Omron CX-Programmer project 新規ﾌﾟﾛｼﾞｪｸﾄ (CX-Programmer 9.34)

# PLC DCS_PLC: CJ2M CPU13
I/O table (CPU CJ2M-CPU13): rack 0 slot 0 CJ1W-CLK23; rack 0 slot 1 CJ1W-SCU21-V1; rack 0 slot 2 CJ1W-OD211

## Global symbols (name address type ; comment)
0.05 BOOL  ; error_clear_sw
12 CHANNEL  ; CH1PV１次1,2桁目
1534.06 BOOL  ; P1受信完了ﾌﾗｸﾞ
1544.06 BOOL  ; P2受信完了ﾌﾗｸﾞ
1559.05 BOOL  ; TXDU命令実行中ﾌﾗｸﾞ
1634.06 BOOL  ; -
2.10 BOOL  ; lot_trace_camera_out1
2.11 BOOL  ; lot_trace_camera_out2
2.12 BOOL  ; lot_trace_camera_out3
2.13 BOOL  ; lot_trace_camera_out4
3000.01 BOOL  ; 送り
3000.02 BOOL  ; 全検査完了
3000.03 BOOL  ; 装置再投入フラグ
3010.01 BOOL  ; ﾗﾝﾆﾝｸﾞ_disable
3010.02 BOOL  ; 耐圧CC_disable
3010.03 BOOL  ; 耐圧CF_disable
3010.04 BOOL  ; 有負荷disable
3010.05 BOOL  ; ｲﾝﾊﾟﾙｽ_disable
3010.06 BOOL  ; ｵﾌﾊﾞｳﾝｽ_disable
3010.07 BOOL  ; RT_disable
3010.08 BOOL  ; MVD_disable
3020.06 BOOL  ; R1_OK
3020.07 BOOL  ; R2_OK
3020.08 BOOL  ; R3_OK
3020.09 BOOL  ; R4_OK
3020.10 BOOL  ; R5_OK
3020.11 BOOL  ; R6_OK
3020.12 BOOL  ; R7_OK
3020.13 BOOL  ; R8_OK
3020.14 BOOL  ; R9_OK
3020.15 BOOL  ; R10_OK
3021.00 BOOL  ; 耐圧CC_OK
3021.01 BOOL  ; 耐圧CF_OK
3021.02 BOOL  ; ｲﾝﾊﾟﾙｽ_OK
3021.03 BOOL  ; 有負荷_OK
3021.04 BOOL  ; ｵﾌﾊﾞｳﾝｽ_OK
3021.05 BOOL  ; RT_OK
3021.06 BOOL  ; MVD_OK
3022.06 BOOL  ; R1_NG
3022.07 BOOL  ; R2_NG
3022.08 BOOL  ; R3_NG
3022.09 BOOL  ; R4_NG
3022.10 BOOL  ; R5_NG
3022.11 BOOL  ; R6_NG
3022.12 BOOL  ; R7_NG
3022.13 BOOL  ; R8_OK
3022.14 BOOL  ; R9_OK
3022.15 BOOL  ; R10_OK
3023.00 BOOL  ; 耐圧CC_OK
3023.01 BOOL  ; 耐圧CF_OK
3023.02 BOOL  ; ｲﾝﾊﾟﾙｽ_OK
3023.03 BOOL  ; 有負荷_OK
3023.04 BOOL  ; ｵﾌﾊﾞｳﾝｽ_OK
3023.05 BOOL  ; RT_OK
3023.06 BOOL  ; MVD_OK
3024.00 BOOL  ; R1
3024.01 BOOL  ; R2
3024.02 BOOL  ; R3
3024.03 BOOL  ; R4
3024.04 BOOL  ; R5
3024.05 BOOL  ; R6
3024.06 BOOL  ; R7
3024.07 BOOL  ; R8
3024.08 BOOL  ; R9
3024.09 BOOL  ; ﾗﾝﾆﾝｸﾞ
3024.10 BOOL  ; 耐圧C-F
3024.11 BOOL  ; 耐圧C-C
3024.12 BOOL  ; ｺｲﾙｲﾝﾊﾟﾙｽ
3024.13 BOOL  ; 有負荷ﾗﾝﾆﾝｸﾞ
3024.14 BOOL  ; ｵﾌﾊﾞｳﾝｽ
3024.15 BOOL  ; CIR
3025.00 BOOL  ; PV-H
3025.01 BOOL  ; PV-L
3025.02 BOOL  ; DV-H
3025.03 BOOL  ; DV-L
3025.04 BOOL  ; TSO
3025.05 BOOL  ; MVD
3050.00 BOOL  ; Ready_RT
3050.01 BOOL  ; Ready_CP
3100.00 BOOL  ; ﾃﾞｰﾀ収集Home
3100.01 BOOL  ; ﾃﾞｰﾀ収集FULL
3100.02 BOOL  ; ﾃﾞｰﾀ収集Ready
3100.03 BOOL  ; CP繰返測定モード
3228 CHANNEL  ; Z2_Target_position
3328 CHANNEL  ; Z2_Now_position
4.14 BOOL  ; lot_trace_camera_out
5000.00 BOOL  ; ﾃﾞｰﾀ収集PLC原点OK
5000.01 BOOL  ; ﾃﾞｰﾀﾊﾞｯﾌｧｰFull
5000.02 BOOL  ; ﾃﾞｰﾀ収集Ready
500.01 BOOL  ; 取出
902.11 BOOL  ; tp_delate_sw
902.12 BOOL  ; tp_all_delete_yes_sw
A202.00 BOOL  ; ﾈｯﾄﾜｰｸ通信命令実行可ﾌﾗｸﾞ
A351 CHANNEL  ; 分秒
A352 CHANNEL  ; 日時
A353 CHANNEL  ; 年月
A356.05 BOOL  ; PORT1送信ﾚﾃﾞｲﾌﾗｸﾞ
A392.05 BOOL  ; RS232Cﾎﾟｰﾄ送信ﾚﾃﾞｲﾌﾗｸﾞ
D0 CHANNEL  ; PC心拍数
D1 CHANNEL  ; PC心拍ﾃﾞｸﾘﾒﾝﾄ用ﾌﾟﾘｽｹｰﾗ
D10 CHANNEL  ; 結果ﾃﾞｰﾀ
D100 CHANNEL  ; 受信CH1PV1,2桁
D1000 CHANNEL  ; １ﾊﾞｲﾄ目
D10000 CHANNEL  ; 1ST
D10000.00 BOOL  ; 搬送送りﾄﾘｶﾞ
D10001.00 BOOL  ; 搬送RT1検査実施
D10001.01 BOOL  ; 搬送RT2検査実施
D10001.02 BOOL  ; 搬送RT3検査実施
D10001.03 BOOL  ; 搬送CP1検査実施
D10001.04 BOOL  ; 搬送CP2検査実施
D10001.05 BOOL  ; 搬送CP3検査実施
D10002.00 BOOL  ; 搬送検査ﾄﾘｶﾞ
D1000.00 BOOL  ; 搬送PLCﾃﾞｰﾀ出力ﾄﾘｶﾞ
D10010 CHANNEL  ; PF_Ch1OVL
D10011 CHANNEL  ; PF_Ch1OVR
D10012 CHANNEL  ; PV_IN
D10014 CHANNEL  ; DV_IN
D10016 CHANNEL  ; CIR_IN
D10018 CHANNEL  ; TSO_IN
D10028 CHANNEL  ; NC_IN
D10030 CHANNEL  ; NO_IN
D10032 CHANNEL  ; CG_IN
D10040 CHANNEL  ; PF_Ch3TOL
D10041 CHANNEL  ; PF_Ch3TOR
D101 CHANNEL  ; 受信CH1PV3,4桁
D10128 CHANNEL  ; NC_IN
D10130 CHANNEL  ; NO_IN
D10132 CHANNEL  ; CG_IN
D102 CHANNEL  ; 受信CH1PV5桁目と小数点
D10200 CHANNEL  ; 3ST
D10202 CHANNEL  ; R2_IN
D10212 CHANNEL  ; PV_OUT
D10214 CHANNEL  ; DV_OUT
D10216 CHANNEL  ; CIR_OUT
D10218 CHANNEL  ; TSO_OUT
D10228 CHANNEL  ; NC_IN
D10230 CHANNEL  ; NO_IN
D10232 CHANNEL  ; CG_OUT
D103 CHANNEL  ; 受信CH1PV6,7桁目
D10300 CHANNEL  ; 4ST
D10303 CHANNEL  ; R3_IN
D10312 CHANNEL  ; PV_OUT
D10314 CHANNEL  ; DV_OUT
D10316 CHANNEL  ; CIR_OUT
D10318 CHANNEL  ; TSO_OUT
D10328 CHANNEL  ; NC_OUT
D10330 CHANNEL  ; NO_OUT
D10332 CHANNEL  ; CG_OUT
D104 CHANNEL  ; 受信CH1DVt,1桁目
D10400 CHANNEL  ; 5ST
D10404 CHANNEL  ; R4_IN
D10412 CHANNEL  ; PV_OUT
D10414 CHANNEL  ; DV_OUT
D10416 CHANNEL  ; CIR_OUT
D10418 CHANNEL  ; TSO_OUT
D10428 CHANNEL  ; NC_OUT
D10430 CHANNEL  ; NO_OUT
D10432 CHANNEL  ; CG_OUT
D105 CHANNEL  ; 受信CH1DV2,3桁目
D10500 CHANNEL  ; 6ST
D10505 CHANNEL  ; R5_IN
D106 CHANNEL  ; 受信CH1DV4,5桁目
D10600 CHANNEL  ; 7ST
D107 CHANNEL  ; 受信CH1DV小数点と6桁目
D10700 CHANNEL  ; 8ST
D10707 CHANNEL  ; 耐圧CC_IN
D108 CHANNEL  ; 受信CH1DV7桁目とt
D10800 CHANNEL  ; 9ST
D10808 CHANNEL  ; 耐圧CF_IN
D109 CHANNEL  ; 受信CH1ｺｲﾙR1,2桁目
D10900 CHANNEL  ; 10ST
D10909 CHANNEL  ; ｲﾝﾊﾟﾙｽIN
D110 CHANNEL  ; 受信CH1ｺｲﾙR3,4桁目
D1100 CHANNEL  ; 結果
D11000 CHANNEL  ; 送信ｴﾘｱ収集PLC
D11010 CHANNEL  ; 有負荷IN
D111 CHANNEL  ; 受信CH1ｺｲﾙR5,6桁目
D11100 CHANNEL  ; 12ST
D11111 CHANNEL  ; ｵﾌﾊﾞｳﾝｽ_IN
D112 CHANNEL  ; 受信CH1ｺｲﾙR小数点,7桁目
D11200 CHANNEL  ; 13ST
D11212 CHANNEL  ; PV_IN
D11214 CHANNEL  ; DV_IN
D11216 CHANNEL  ; CIR_IN
D11218 CHANNEL  ; TSO_IN
D11228 CHANNEL  ; MVD_IN
D11300 CHANNEL  ; 14ST
D11328 CHANNEL  ; MVD_IN
D114 CHANNEL  ; 受信CH1TSO2,3桁目
D11400 CHANNEL  ; 15ST
D115 CHANNEL  ; 受信CH1TSO4,5桁目
D11500 CHANNEL  ; 16ST
D11531 CHANNEL  ; R6_IN
D116 CHANNEL  ; 受信CH1TSO小数点6桁目
D11600 CHANNEL  ; 17ST
D11632 CHANNEL  ; R7_IN
D117 CHANNEL  ; 受信CH1TSO7桁目,t
D11700 CHANNEL  ; 18ST
D11733 CHANNEL  ; R8_IN
D11800 CHANNEL  ; 19ST
D11834 CHANNEL  ; R9_IN
D11900 CHANNEL  ; 20ST
D11935 CHANNEL  ; R10_IN
D11996.00 BOOL  ; 収集PLCﾃﾞｰﾀ満杯
D11997.00 BOOL  ; PC起動OKﾌﾗｸﾞ
D11998 CHANNEL  ; PC読込許可ﾌﾗｸﾞ
D11999 CHANNEL  ; PC読込完了ﾌﾗｸﾞｸﾘｱ依頼
D12000 CHANNEL  ; PC読込完了ﾌﾗｸﾞ
D12001.00 BOOL  ; PC起動中Pulse
D12100 CHANNEL  ; 22ST
D12200 CHANNEL  ; 23ST
D12212 CHANNEL  ; PV_OUT
D12300 CHANNEL  ; 24ST
D12400 CHANNEL  ; 25ST
D12401 CHANNEL  ; R1_OUT
D12402 CHANNEL  ; R2_OUT
D12403 CHANNEL  ; R3_OUT
D12404 CHANNEL  ; R4_OUT
D12405 CHANNEL  ; R5_OUT
D12407 CHANNEL  ; 耐圧CC_OUT
D12408 CHANNEL  ; 耐圧CF_OUT
D12409 CHANNEL  ; ｲﾝﾊﾟﾙｽOUT
D12410 CHANNEL  ; 有負荷OUT
D12411 CHANNEL  ; ｵﾌﾊﾞｳﾝｽ_OUT
D12412 CHANNEL  ; PV_OUT
D12414 CHANNEL  ; DV_OUT
D12416 CHANNEL  ; CIR_OUT
D12418 CHANNEL  ; TSO_OUT
D12428 CHANNEL  ; MVD_OUT
D12431 CHANNEL  ; R6_OUT
D12432 CHANNEL  ; R7_OUT
D12433 CHANNEL  ; R8_OUT
D12434 CHANNEL  ; R9_OUT
D12435 CHANNEL  ; R10_OUT
D12500 CHANNEL  ; 26ST
D12600 CHANNEL  ; 27ST
D12700 CHANNEL  ; 28ST
D12701 CHANNEL  ; R1_OUT
D12702 CHANNEL  ; R2_OUT
D12703 CHANNEL  ; R3_OUT
D12704 CHANNEL  ; R4_OUT
D12705 CHANNEL  ; R5_OUT
D12707 CHANNEL  ; 耐圧CC_OUT
D12708 CHANNEL  ; 耐圧CF_OUT
D12709 CHANNEL  ; ｲﾝﾊﾟﾙｽOUT
D12710 CHANNEL  ; 有負荷OUT
D12711 CHANNEL  ; ｵﾌﾊﾞｳﾝｽOUT
D12712 CHANNEL  ; PV_OUT
D12714 CHANNEL  ; DV_OUT
D12716 CHANNEL  ; CIR_OUT
D12718 CHANNEL  ; TSO_OUT
D12728 CHANNEL  ; MVD_OUT
D12730 CHANNEL  ; NO_OUT
D12731 CHANNEL  ; R6_OUT
D12732 CHANNEL  ; R7_OUT
D12733 CHANNEL  ; R8_OUT
D12734 CHANNEL  ; R9_OUT
D12735 CHANNEL  ; R10_OUT
D13000 CHANNEL  ; TMP有無
D13001 CHANNEL  ; TMP分秒
D13002 CHANNEL  ; TMP日時
D13003 CHANNEL  ; TMP年月
D13004 CHANNEL  ; TMP順番
D13005 CHANNEL  ; TMPﾁｬﾝﾈﾙ
D13006 CHANNEL  ; TMPﾁｬﾝﾈﾙ
D13007 CHANNEL  ; TMP機種コード
D13008 CHANNEL  ; TMP機種名
D13018 CHANNEL  ; TMP再投入
D13019 CHANNEL  ; PV_TMP
D13021 CHANNEL  ; DV_TMP
D13023 CHANNEL  ; TSO_TMP
D13025 CHANNEL  ; NC_TMP
D13027 CHANNEL  ; NO_TMP
D13029 CHANNEL  ; CG_TMP
D13031 CHANNEL  ; PV_TMP
D13033 CHANNEL  ; DV_TMP
D13035 CHANNEL  ; TSO_TMP
D13037 CHANNEL  ; CIR_TMP
D13039 CHANNEL  ; MVD_TMP
D13041 CHANNEL  ; 有負荷R_TMP
D13042 CHANNEL  ; 耐圧C-F_TMP
D13043 CHANNEL  ; 耐圧C-C_TMP
D13044 CHANNEL  ; ｵﾌﾊﾞｳﾝｽ_TMP
D13045 CHANNEL  ; ｲﾝﾊﾟﾙｽ_TMP
D13046 CHANNEL  ; ﾗﾝﾆﾝｸﾞ_TMP
D13047 CHANNEL  ; TMP判定
D13050 CHANNEL  ; PV_TMP
D13052 CHANNEL  ; DV_TMP
D13054 CHANNEL  ; TSO_TMP
D13056 CHANNEL  ; CIR_TMP
D13058 CHANNEL  ; NC_MVD_TMP
D13060 CHANNEL  ; NO_TMP
D13062 CHANNEL  ; CG_IN
D13063 CHANNEL  ; 有負荷_TMP
D13064 CHANNEL  ; 耐圧CC_TMP
D13065 CHANNEL  ; 耐圧CF_TMP
D13066 CHANNEL  ; ｵﾌﾊﾞｳﾝｽ_TMP
D13067 CHANNEL  ; ｲﾝﾊﾟﾙｽ_TMP
D13068 CHANNEL  ; R1TMP
D13069 CHANNEL  ; R2_TMP
D13070 CHANNEL  ; R3_TMP
D13071 CHANNEL  ; R4_TMP
D13072 CHANNEL  ; R5_TMP
D13073 CHANNEL  ; R6_TMP
D13074 CHANNEL  ; R7_TMP
D13075 CHANNEL  ; R8_TMP
D13076 CHANNEL  ; R9_TMP
D13077 CHANNEL  ; R10_TMP
D13078 CHANNEL  ; RT_TMP
D13079 CHANNEL  ; MVD_TMP
D13100 CHANNEL  ; PC書込中フラグ
D13102 CHANNEL  ; ﾃﾞﾊﾞｯｸﾞ用カウンタ
D13200 CHANNEL  ; Dｴﾘｱｸﾘｱﾎﾟｲﾝﾀ
D13300 CHANNEL  ; ｺﾝﾄﾛｰﾙﾃﾞｰﾀ1-1
D13301 CHANNEL  ; ｺﾝﾄﾛｰﾙﾃﾞｰﾀ1-2
D13302 CHANNEL  ; ｺﾝﾄﾛｰﾙﾃﾞｰﾀ2-1
D13303 CHANNEL  ; ｺﾝﾄﾛｰﾙﾃﾞｰﾀ2-2
D13400 CHANNEL  ; RT受信ﾃﾞｰﾀ1
D13402 CHANNEL  ; RT受信ﾃﾞｰﾀPV3
D13403 CHANNEL  ; RT受信ﾃﾞｰﾀ2
D13404 CHANNEL  ; RT受信ﾃﾞｰﾀDV4
D13405 CHANNEL  ; RT受信ﾃﾞｰﾀDV1
D13406 CHANNEL  ; RT受信ﾃﾞｰﾀ3
D13407 CHANNEL  ; RT受信ﾃﾞｰﾀDV3
D13408 CHANNEL  ; RT受信ﾃﾞｰﾀDV3
D13409 CHANNEL  ; RT受信ﾃﾞｰﾀ4
D13410 CHANNEL  ; RT受信ﾃﾞｰﾀCI2
D13411 CHANNEL  ; RT受信ﾃﾞｰﾀCI3
D13412 CHANNEL  ; RT受信ﾃﾞｰﾀ5
D13414 CHANNEL  ; RT受信ﾃﾞｰﾀTSO1
D13415 CHANNEL  ; RT受信ﾃﾞｰﾀ6
D13416 CHANNEL  ; RT受信ﾃﾞｰﾀTSO3
D13417 CHANNEL  ; RT受信ﾃﾞｰﾀTSO4
D13450 CHANNEL  ; RT_OVL
D13452 CHANNEL  ; RT_OVR
D13453 CHANNEL  ; PV1次4
D13454 CHANNEL  ; RT_RVL
D13455 CHANNEL  ; DV1次1
D13456 CHANNEL  ; RT_RVR
D13457 CHANNEL  ; DV1次3
D13458 CHANNEL  ; DV1次4
D13460 CHANNEL  ; CP_Ch1NCL
D13461 CHANNEL  ; CI1次2
D13462 CHANNEL  ; CP_Ch1NCR
D13463 CHANNEL  ; CI1次4
D13464 CHANNEL  ; CP_Ch1NOL
D13465 CHANNEL  ; TSO1次1
D13466 CHANNEL  ; CP_Ch1NOR
D13467 CHANNEL  ; TSO1次3
D13468 CHANNEL  ; CP_Ch1CGL
D13469 CHANNEL  ; CI1次5
D13470 CHANNEL  ; CP_Ch1CGR
D13472 CHANNEL  ; CP_Ch2NCL
D13474 CHANNEL  ; CP_Ch2NCR
D13476 CHANNEL  ; CP_Ch2NOL
D13478 CHANNEL  ; CP_Ch2NOR
D13480 CHANNEL  ; CP_Ch2CGL
D13482 CHANNEL  ; CP_Ch2CGR
D13484 CHANNEL  ; CP_Ch3NCL
D13486 CHANNEL  ; CP_Ch3NCR
D13488 CHANNEL  ; CP_Ch3NOL
D13490 CHANNEL  ; CP_Ch3NOR
D13492 CHANNEL  ; CP_Ch3CGL
D13494 CHANNEL  ; CP_Ch3CGR
D13496 CHANNEL  ; RT_TOL
D13498 CHANNEL  ; RT_TOR
D13500 CHANNEL  ; PF_Ch1OVL
D13501 CHANNEL  ; PF_Ch1OVR
D13502 CHANNEL  ; PF_Ch2OVL
D13503 CHANNEL  ; PF_Ch2OVR
D13504 CHANNEL  ; PF_Ch3OVL
D13505 CHANNEL  ; PF_Ch3OVR
D13506 CHANNEL  ; PF_Ch1RVL
D13507 CHANNEL  ; PF_Ch1RVR
D13508 CHANNEL  ; PF_Ch2RVL
D13509 CHANNEL  ; PF_Ch2RVR
D13510 CHANNEL  ; PF_Ch3RVL
D13511 CHANNEL  ; PF_Ch3RVR
D13512 CHANNEL  ; PF_Ch1NCL
D13513 CHANNEL  ; PF_Ch1NCR
D13514 CHANNEL  ; PF_Ch1NOL
D13515 CHANNEL  ; PF_Ch1NOR
D13516 CHANNEL  ; PF_Ch1CGL
D13517 CHANNEL  ; PF_Ch1CGR
D13518 CHANNEL  ; PF_Ch2NCL
D13519 CHANNEL  ; PF_Ch2NCR
D13520 CHANNEL  ; PF_Ch2NOL
D13521 CHANNEL  ; PF_Ch2NOR
D13522 CHANNEL  ; PF_Ch2CGL
D13523 CHANNEL  ; PF_Ch2CGR
D13524 CHANNEL  ; PF_Ch3NCL
D13525 CHANNEL  ; PF_Ch3NCR
D13526 CHANNEL  ; PF_Ch3NOL
D13527 CHANNEL  ; PF_Ch3NOR
D13528 CHANNEL  ; PF_Ch3CGL
D13529 CHANNEL  ; PF_Ch3CGR
D13530 CHANNEL  ; PF_Ch3TOL
D13531 CHANNEL  ; PF_Ch3TOR
D13532 CHANNEL  ; TSO2次3
D13533 CHANNEL  ; TSO2次4
D13550 CHANNEL  ; PV2次TMP1
D13551 CHANNEL  ; PV2次TMP2
D13552 CHANNEL  ; PV2次TMP3
D13553 CHANNEL  ; PV2次TMP4
D13554 CHANNEL  ; PV2次TMP5
D13555 CHANNEL  ; PV2次TMP6
D13556 CHANNEL  ; PV2次TMP7
D13560 CHANNEL  ; DV2次TMP1
D13561 CHANNEL  ; DV2次TMP2
D13562 CHANNEL  ; DV2次TMP3
D13563 CHANNEL  ; DV2次TMP4
D13564 CHANNEL  ; DV2次TMP5
D13565 CHANNEL  ; DV2次TMP6
D13566 CHANNEL  ; DV2次TMP7
D13570 CHANNEL  ; CI2次TMP1
D13571 CHANNEL  ; CI2次TMP2
D13572 CHANNEL  ; CI2次TMP3
D13573 CHANNEL  ; CI2次TMP4
D13574 CHANNEL  ; CI2次TMP5
D13575 CHANNEL  ; CI2次TMP6
D13576 CHANNEL  ; CI2次TMP7
D13580 CHANNEL  ; TSO2次TMP1
D13581 CHANNEL  ; TSO2次TMP2
D13582 CHANNEL  ; TSO2次TMP3
D13583 CHANNEL  ; TSO2次TMP4
D13584 CHANNEL  ; TSO2次TMP5
D13585 CHANNEL  ; TSO2次TMP6
D13586 CHANNEL  ; TSO2次TMP7
D13604 CHANNEL  ; PV
D13610 CHANNEL  ; DV_HEX
D13612 CHANNEL  ; DV_BIN
D13614 CHANNEL  ; DV
D13620 CHANNEL  ; CI_HEX
D13622 CHANNEL  ; CI_BIN
D13624 CHANNEL  ; CIR
D13630 CHANNEL  ; TSO_HEX
D13632 CHANNEL  ; TSO_BIN
D13634 CHANNEL  ; TSO
D13700 CHANNEL  ; CP受信ﾃﾞｰﾀ1
D13702 CHANNEL  ; CP受信ﾃﾞｰﾀ2
D13703 CHANNEL  ; CP受信ﾃﾞｰﾀ2
D13704 CHANNEL  ; CP受信ﾃﾞｰﾀ3
D13706 CHANNEL  ; CP受信ﾃﾞｰﾀ3
D13709 CHANNEL  ; CP受信ﾃﾞｰﾀ4
D13712 CHANNEL  ; CP受信ﾃﾞｰﾀ5
D13714 CHANNEL  ; CP元ﾃﾞｰﾀNCCP
D13715 CHANNEL  ; CP受信ﾃﾞｰﾀ6
D13717 CHANNEL  ; CP元ﾃﾞｰﾀNOCP
D13718 CHANNEL  ; CP受信ﾃﾞｰﾀ7
D13720 CHANNEL  ; CP元ﾃﾞｰﾀCG
D13721 CHANNEL  ; CP受信ﾃﾞｰﾀ8
D13724 CHANNEL  ; CP受信ﾃﾞｰﾀ9
D13727 CHANNEL  ; CP受信ﾃﾞｰﾀ10
D13730 CHANNEL  ; CP受信ﾃﾞｰﾀ11
D13733 CHANNEL  ; CP受信ﾃﾞｰﾀ12
D13736 CHANNEL  ; CP受信ﾃﾞｰﾀ13
D13739 CHANNEL  ; CP受信ﾃﾞｰﾀ14
D13742 CHANNEL  ; CP受信ﾃﾞｰﾀ15
D13745 CHANNEL  ; CP受信ﾃﾞｰﾀ16
D13748 CHANNEL  ; CP受信ﾃﾞｰﾀ17
D13751 CHANNEL  ; CP受信ﾃﾞｰﾀ18
D13800 CHANNEL  ; PF_Ch3TOL
D13801 CHANNEL  ; PF_Ch3TOR
D13809 CHANNEL  ; NCCP_TMP1
D13811 CHANNEL  ; NOCP_TMP1
D13813 CHANNEL  ; CG_TMP1
D13859 CHANNEL  ; NCCPTMP2
D13861 CHANNEL  ; NOCP_TMP2
D13863 CHANNEL  ; CG_TMP2
D13904 CHANNEL  ; MVD
D13909 CHANNEL  ; NCCP
D13911 CHANNEL  ; NOCP
D13913 CHANNEL  ; CG
D13920 CHANNEL  ; ch番号
D13922 CHANNEL  ; 機種ｺｰﾄﾞ
D13924 CHANNEL  ; 機種名1/7
D14000 CHANNEL  ; ST0
D14100 CHANNEL  ; ST1
D14200 CHANNEL  ; ST2
D14300 CHANNEL  ; ST3
D14400 CHANNEL  ; ST4
D14500 CHANNEL  ; ST5
D14600 CHANNEL  ; ST6
D150 CHANNEL  ; CH1PV１次ﾃﾞｰﾀ1,2桁目
D151 CHANNEL  ; CH1PV１次ﾃﾞｰﾀ3,4桁目
D152 CHANNEL  ; CH1PV１次5,6桁目
D153 CHANNEL  ; CH1PV１次ﾃﾞｰﾀ7,8桁目
D155 CHANNEL  ; CH1DV１次ﾃﾞｰﾀ1,2桁目
D156 CHANNEL  ; CH1DV１次ﾃﾞｰﾀ3,4桁目
D157 CHANNEL  ; CH1DV１次ﾃﾞｰﾀ5,6桁目
D158 CHANNEL  ; CH1DV１次ﾃﾞｰﾀ7,8桁目
D160 CHANNEL  ; CH1ｺｲﾙR1次ﾃﾞｰﾀ1,2桁目
D161 CHANNEL  ; CH1ｺｲﾙR1次ﾃﾞｰﾀ3,4桁目
D162 CHANNEL  ; CH1ｺｲﾙR1次ﾃﾞｰﾀ5,6桁目
D163 CHANNEL  ; CH1ｺｲﾙR1次ﾃﾞｰﾀ7,8桁目
D165 CHANNEL  ; CH1TSO1次ﾃﾞｰﾀ1,2桁目
D166 CHANNEL  ; CH1TSO1次ﾃﾞｰﾀ3,4桁目
D167 CHANNEL  ; CH1TSO1次ﾃﾞｰﾀ5,6桁目
D168 CHANNEL  ; CH1TSO1次ﾃﾞｰﾀ7,8桁目
D169 CHANNEL  ; CH1ｺｲﾙR1次ﾃﾞｰﾀ小数点,8桁目
D1.02 BOOL  ; PC心拍ﾃﾞｸﾘﾒﾝﾄPulse
D20 CHANNEL  ; ｺﾝﾄﾛｰﾙﾃﾞｰﾀ
D200 CHANNEL  ; CH1PV2次ﾃﾞｰﾀ1,2桁目
D201 CHANNEL  ; CH1PV２次ﾃﾞｰﾀ3,4桁目
D202 CHANNEL  ; CH1PV２次ﾃﾞｰﾀ5,6桁目
D203 CHANNEL  ; CH1PV２次ﾃﾞｰﾀ7,8桁目
D21 CHANNEL  ; ｺﾝﾄﾛｰﾙﾃﾞｰﾀ+1
D210 CHANNEL  ; CH1DV2次ﾃﾞｰﾀ1,2桁目
D211 CHANNEL  ; CH1DV２次ﾃﾞｰﾀ3,4桁目
D212 CHANNEL  ; CH1DV２次ﾃﾞｰﾀ5,6桁目
D213 CHANNEL  ; CH1DV２次ﾃﾞｰﾀ7,8桁目
D22 CHANNEL  ; P2ｺﾝﾄﾛｰﾙﾃﾞｰﾀ
D220 CHANNEL  ; CH1ｺｲﾙR2次ﾃﾞｰﾀ1,2桁目
D221 CHANNEL  ; CH1ｺｲﾙR2次ﾃﾞｰﾀ3,4桁目
D222 CHANNEL  ; CH1ｺｲﾙR2次ﾃﾞｰﾀ5,6桁目
D223 CHANNEL  ; CH1ｺｲﾙR2次ﾃﾞｰﾀ7,8桁目
D23 CHANNEL  ; P2ｺﾝﾄﾛｰﾙﾃﾞｰﾀ+1
D230 CHANNEL  ; CH1TSO2次ﾃﾞｰﾀ1,2桁目
D231 CHANNEL  ; CH1TSO2次ﾃﾞｰﾀ3,4桁目
D232 CHANNEL  ; CH1TSO2次ﾃﾞｰﾀ5,6桁目
D233 CHANNEL  ; CH1TSO2次ﾃﾞｰﾀ7,8桁目
D250 CHANNEL  ; CH1PV１次2桁目
D251 CHANNEL  ; CH1PV１次３桁目
D252 CHANNEL  ; CH1PV１次４桁目
D253 CHANNEL  ; CH1PV１次５桁目
D254 CHANNEL  ; CH1PV１次６桁目
D255 CHANNEL  ; CH1PV１次７桁目
D256 CHANNEL  ; CH1PV１次８桁目
D260 CHANNEL  ; CH1DV１次2桁目
D261 CHANNEL  ; CH1DV１次３桁目
D262 CHANNEL  ; CH1DV１次４桁目
D263 CHANNEL  ; CH1DV１次５桁目
D264 CHANNEL  ; CH1DV１次６桁目
D265 CHANNEL  ; CH1DV１次７桁目
D266 CHANNEL  ; CH1DV１次８桁目
D270 CHANNEL  ; CH1ｺｲﾙR1次2桁目
D271 CHANNEL  ; CH1ｺｲﾙR1次3桁目
D272 CHANNEL  ; CH1ｺｲﾙR1次4桁目
D274 CHANNEL  ; CH1ｺｲﾙR1次6桁目
D275 CHANNEL  ; CH1ｺｲﾙR1次7桁目
D276 CHANNEL  ; CH1ｺｲﾙR1次8桁目
D280 CHANNEL  ; CH1TSO1次2桁目
D281 CHANNEL  ; CH1TSO1次3桁目
D282 CHANNEL  ; CH1TSO1次4桁目
D284 CHANNEL  ; CH1TSO1次6桁目
D285 CHANNEL  ; CH1TSO1次7桁目
D286 CHANNEL  ; CH1TSO1次8桁目
D300 CHANNEL  ; CH1PV１６進
D302 CHANNEL  ; CH1PV１０進
D304 CHANNEL  ; CH1PV
D310 CHANNEL  ; CH1DV１６進
D312 CHANNEL  ; CH1DV１０進
D314 CHANNEL  ; CH1DV
D320 CHANNEL  ; CH1ｺｲﾙR１６進
D322 CHANNEL  ; CH1ｺｲﾙR１０進
D324 CHANNEL  ; CH1CIR
D330 CHANNEL  ; CH1TSO１６進
D332 CHANNEL  ; CH1TSO１０進
D334 CHANNEL  ; CH1TSO
D400 CHANNEL  ; MVD受信元ﾃﾞｰﾀ
D403 CHANNEL  ; CP元ﾃﾞｰﾀ機種ｺｰﾄﾞ
D406 CHANNEL  ; CP元ﾃﾞｰﾀ機種名1/7
D414 CHANNEL  ; CP元ﾃﾞｰﾀNCCP
D417 CHANNEL  ; CP元ﾃﾞｰﾀNOCP
D420 CHANNEL  ; CP元ﾃﾞｰﾀCG
D480 CHANNEL  ; tmp1
D481 CHANNEL  ; tmp2
D50 CHANNEL  ; 結果ﾃﾞｰﾀ
D500 CHANNEL  ; ch番号
D501 CHANNEL  ; 機種ｺｰﾄﾞ
D502 CHANNEL  ; 機種名1/7
D509 CHANNEL  ; NCCP
D511 CHANNEL  ; NOCP
D513 CHANNEL  ; CG
D560 CHANNEL  ; -
D630 CHANNEL  ; -
D632 CHANNEL  ; -
D800 CHANNEL  ; PC_Lot1Product
D810 CHANNEL  ; PC_Lot2Product
D820 CHANNEL  ; PC_Lo3Product
D860 CHANNEL  ; PC_Lot1Quantity
D861 CHANNEL  ; PC_Lot2Quantity
D862 CHANNEL  ; PC_Lot3Quantity
D863 CHANNEL  ; -
D864 CHANNEL  ; -
D866 CHANNEL  ; -
D867 CHANNEL  ; -
D868 CHANNEL  ; -
D875 CHANNEL  ; -
D876 CHANNEL  ; -
D877 CHANNEL  ; -
D878 CHANNEL  ; -
D879 CHANNEL  ; -
D881 CHANNEL  ; -
D882 CHANNEL  ; -
D910 CHANNEL  ; tp_program_number
E0 CHANNEL  ; 本体PLC測定順番
E110 CHANNEL  ; 分秒ﾃﾞｰﾀ
E11000 CHANNEL  ; ｽﾀｯｸNo91
E111 CHANNEL  ; 日時ﾃﾞｰﾀ
E112 CHANNEL  ; 年月ﾃﾞｰﾀ
E13 CHANNEL  ; 本体PLC ch番号
E14 CHANNEL  ; 再投入
E1800 CHANNEL  ; ﾃﾞｰﾀ収集パソコンOK
E1802 CHANNEL  ; PC_First_cycle_Flag
E1803 CHANNEL  ; PC_Stac_Clear_Flag
E1810 CHANNEL  ; 分秒ﾃﾞｰﾀ
E1811 CHANNEL  ; ｼﾌﾄ中
E1812 CHANNEL  ; 年月データ
E1820 CHANNEL  ; 本体ﾃﾞｰﾀ有通信用
E1821 CHANNEL  ; ｼﾌﾄ中
E1822 CHANNEL  ; クリア先頭番地
E1830 CHANNEL  ; サーチ中番地
E1832 CHANNEL  ; 転送先番地
E1900 CHANNEL  ; 元ﾃﾞｰﾀ有無
E1904 CHANNEL  ; PC順番
E1906 CHANNEL  ; PCﾁｬﾝﾈﾙ
E1907 CHANNEL  ; PC機種コード
E1908 CHANNEL  ; PC機種名
E1918 CHANNEL  ; PC再投入
E1919 CHANNEL  ; 元PVﾃﾞｰﾀ
E1921 CHANNEL  ; 元DVﾃﾞｰﾀ
E1923 CHANNEL  ; 元TSOﾃﾞｰﾀ
E1925 CHANNEL  ; 元NCﾃﾞｰﾀ
E1927 CHANNEL  ; 元NOﾃﾞｰﾀ
E1929 CHANNEL  ; 元CGﾃﾞｰﾀ
E1931 CHANNEL  ; CH_PV
E1933 CHANNEL  ; CH_DV
E1935 CHANNEL  ; CH_TSO
E1937 CHANNEL  ; CH_CIR
E1939 CHANNEL  ; CH_MVD
E1941 CHANNEL  ; 有負荷
E1942 CHANNEL  ; 耐圧CC
E1943 CHANNEL  ; 耐圧CF
E1944 CHANNEL  ; ｵﾌﾊﾞｳﾝｽ
E1945 CHANNEL  ; ｲﾝﾊﾟﾙｽ
E1946 CHANNEL  ; ﾗﾝﾆﾝｸﾞ
E1947 CHANNEL  ; PC判定
E1950 CHANNEL  ; 本体データ有(仮PCダミー)
E2 CHANNEL  ; 本体PLC機種ｺｰﾄﾞ
E2000 CHANNEL  ; ｽﾀｯｸｴﾘｱ先頭
E2050 CHANNEL  ; ﾃﾞｰﾀ有無2番目
E2100 CHANNEL  ; ﾃﾞｰﾀ有無2番目
E3 CHANNEL  ; 本体PLC機種名
E32000 CHANNEL  ; -
E32001 CHANNEL  ; -
E32002 CHANNEL  ; -
E32011 CHANNEL  ; -
E32012 CHANNEL  ; -
E32013 CHANNEL  ; -
E32200 CHANNEL  ; -
E32201 CHANNEL  ; -
E32202 CHANNEL  ; -
E32203 CHANNEL  ; -
E32204 CHANNEL  ; -
E32205 CHANNEL  ; -
E32206 CHANNEL  ; -
E32207 CHANNEL  ; -
E32208 CHANNEL  ; -
E32209 CHANNEL  ; -
E32210 CHANNEL  ; -
E32300 CHANNEL  ; -
E32301 CHANNEL  ; 分秒先
E32302 CHANNEL  ; 日時先
E32303 CHANNEL  ; 年月先
E32304 CHANNEL  ; 収集PLC順番
E32305 CHANNEL  ; -
E32306 CHANNEL  ; 収集PLCﾁｬﾝﾈﾙ
E32307 CHANNEL  ; 収集PLC機種コード
E32308 CHANNEL  ; 収集PLC機種名
E32309 CHANNEL  ; -
E32315 CHANNEL  ; -
E32318 CHANNEL  ; 収集PLC再投入
E32319 CHANNEL  ; -
E32320 CHANNEL  ; -
E32330 CHANNEL  ; -
E32340 CHANNEL  ; -
E32347 CHANNEL  ; 収集PLC判定
E32349 CHANNEL  ; -
E32400 CHANNEL  ; -
E32401 CHANNEL  ; -
E32515 CHANNEL  ; -
E32517 CHANNEL  ; -
E32600 CHANNEL  ; -
E32601 CHANNEL  ; -
E32610 CHANNEL  ; -
E32620 CHANNEL  ; -
E32630 CHANNEL  ; -
E32640 CHANNEL  ; -
E32641 CHANNEL  ; -
E50 CHANNEL  ; -
E6950 CHANNEL  ; ｽﾀｯｸｆｕｌｌ
E9900 CHANNEL  ; スタックFull
T0000 BOOL  ; ﾌﾞﾛｯｸ転送完了待ち時間
T0990 BOOL  ; -
T0991 BOOL  ; -
T0992 BOOL  ; -
T0993 BOOL  ; -
T0994 BOOL  ; -
T0995 BOOL  ; -
T0996 BOOL  ; -
W100.00 BOOL  ; 検査終了入力
W100.01 BOOL  ; RT収集S/C
W100.02 BOOL  ; RT収集S/C終了
W100.03 BOOL  ; RTﾃﾞｰﾀ有
W100.04 BOOL  ; 転送ｴﾘｱｸﾘｱ完
W100.05 BOOL  ; RTﾃﾞｰﾀ取得済
W101.00 BOOL  ; CP検査終了入力
W101.01 BOOL  ; CP収集S/C
W101.02 BOOL  ; CP収集S/C終了
W101.03 BOOL  ; CPﾃﾞｰﾀ有
W101.04 BOOL  ; 転送ｴﾘｱｸﾘｱ完
W101.05 BOOL  ; CPﾃﾞｰﾀ取得済
W102.05 BOOL  ; OkNgﾃﾞｰﾀ取得済
W103.00 BOOL  ; RT1検査実施ﾌﾗｸﾞ
W103.01 BOOL  ; RT2検査実施ﾌﾗｸﾞ
W103.02 BOOL  ; RT3検査実施ﾌﾗｸﾞ
W103.03 BOOL  ; CP1検査実施ﾌﾗｸﾞ
W103.04 BOOL  ; CP2検査実施ﾌﾗｸﾞ
W103.05 BOOL  ; CP3検査実施ﾌﾗｸﾞ
W110.01 BOOL  ; RT転送開始
W110.02 BOOL  ; RT転送完了
W111.01 BOOL  ; MVD転送開始
W111.02 BOOL  ; CP受信完了
W120.00 BOOL  ; CH1PVPBｺｰﾄﾞｾｯﾄ完了
W120.01 BOOL  ; CH1PVORｺｰﾄﾞｾｯﾄ完了
W120.02 BOOL  ; CH1PVNCｺｰﾄﾞｾｯﾄ完了
W120.03 BOOL  ; CH1PVADｺｰﾄﾞｾｯﾄ完了
W120.04 BOOL  ; CH1PVMDｺｰﾄﾞｾｯﾄ完了
W120.05 BOOL  ; CH1PVLMｺｰﾄﾞｾｯﾄ完了
W120.10 BOOL  ; CH1PV測定ﾐｽｺｰﾄﾞｾｯﾄ完了
W120.11 BOOL  ; CH1PVﾃﾞｰﾀ入れ替え
W120.12 BOOL  ; CH1PVﾃﾞｰﾀ入れ替え完了
W130.00 BOOL  ; CH1DVPBｺｰﾄﾞｾｯﾄ完了
W130.01 BOOL  ; CH1DVORｺｰﾄﾞｾｯﾄ完了
W130.02 BOOL  ; CH1DVNCｺｰﾄﾞｾｯﾄ完了
W130.03 BOOL  ; CH1DVADｺｰﾄﾞｾｯﾄ完了
W130.04 BOOL  ; CH1DVMDｺｰﾄﾞｾｯﾄ完了
W130.05 BOOL  ; CH1DVLMｺｰﾄﾞｾｯﾄ完了
W130.10 BOOL  ; CH1DV測定ﾐｽｺｰﾄﾞｾｯﾄ完了
W130.11 BOOL  ; CH1DVﾃﾞｰﾀ入れ替え
W130.12 BOOL  ; CH1DVﾃﾞｰﾀ入れ替え完了
W140.00 BOOL  ; CH1ｺｲﾙRPBｺｰﾄﾞｾｯﾄ完了
W140.01 BOOL  ; CH1ｺｲﾙRORｺｰﾄﾞｾｯﾄ完了
W140.02 BOOL  ; CH1ｺｲﾙRNCｺｰﾄﾞｾｯﾄ完了
W140.03 BOOL  ; CH1ｺｲﾙRADｺｰﾄﾞｾｯﾄ完了
W140.04 BOOL  ; CH1ｺｲﾙRMDｺｰﾄﾞｾｯﾄ完了
W140.05 BOOL  ; CH1ｺｲﾙRLMｺｰﾄﾞｾｯﾄ完了
W140.10 BOOL  ; CH1ｺｲﾙR測定ﾐｽｺｰﾄﾞｾｯﾄ完了
W140.11 BOOL  ; CH1ｺｲﾙRﾃﾞｰﾀ入れ替え
W140.12 BOOL  ; CH1ｺｲﾙRﾃﾞｰﾀ入れ替え完了
W150.00 BOOL  ; CH1TSOPBｺｰﾄﾞｾｯﾄ完了
W150.01 BOOL  ; CH1TSOORｺｰﾄﾞｾｯﾄ完了
W150.02 BOOL  ; CH1TSONCｺｰﾄﾞｾｯﾄ完了
W150.03 BOOL  ; CH1TSOADｺｰﾄﾞｾｯﾄ完了
W150.04 BOOL  ; CH1TSOMDｺｰﾄﾞｾｯﾄ完了
W150.05 BOOL  ; CH1TSOOLMｺｰﾄﾞｾｯﾄ完了
W150.10 BOOL  ; CH1TSO測定ﾐｽｺｰﾄﾞｾｯﾄ完了
W150.11 BOOL  ; CH1TSOﾃﾞｰﾀ入れ替え
W150.12 BOOL  ; CH1TSOﾃﾞｰﾀ入れ替え完了
W15.00 BOOL  ; terminal1_put_ok
W15.01 BOOL  ; terminal2_put_ok
W15.02 BOOL  ; restart_sw
W15.03 BOOL  ; PC_lot_data_setting_ok
W15.04 BOOL  ; fail_box_det1
W200.00 BOOL  ; 受信開始
W200.01 BOOL  ; ｼﾌﾄ中
W200.02 BOOL  ; ｼﾌﾄ終了
W300.00 BOOL  ; ｽﾀｯｸ書込み開始
W300.01 BOOL  ; 読込中
W300.02 BOOL  ; 読込終了
W300.03 BOOL  ; ｽﾀｯｸ転送開始
W300.04 BOOL  ; 空きサーチ開始
W300.05 BOOL  ; 空きサーチ完了
W300.06 BOOL  ; スタック転送完了
W301.00 BOOL  ; ALLﾃﾞｰﾀｸﾘｱ_ﾄﾘｶﾞ
W301.01 BOOL  ; クリア開始
W301.02 BOOL  ; クリア完
W301.03 BOOL  ; PLCﾊﾝﾄﾞｼｪｲｸ初期化
W302.00 BOOL  ; ｼﾌﾄ開始
W302.01 BOOL  ; ｼﾌﾄ完
W302.02 BOOL  ; PC読込完了
W302.03 BOOL  ; PCﾊﾝﾄﾞｼｪｲｸ完了
W302.04 BOOL  ; ﾌﾞﾛｯｸ転送完了待ち
W302.05 BOOL  ; PC読込完了ﾌﾗｸﾞｸﾘｱ待ち
W310.00 BOOL  ; RT書込み開始
W310.01 BOOL  ; RT書込み完
W310.08 BOOL  ; MVD書込み開始
W310.09 BOOL  ; MVD書込み完
W311.00 BOOL  ; ｼﾌﾄ開始
W311.01 BOOL  ; ｼﾌﾄ完
W311.02 BOOL  ; データ揃ったよ
W311.03 BOOL  ; chk1
W311.04 BOOL  ; chk2
W311.05 BOOL  ; chk3
W311.06 BOOL  ; chk4
W311.07 BOOL  ; chk5
W311.08 BOOL  ; chk6
W311.09 BOOL  ; chk7
W311.10 BOOL  ; chk8
W312.00 BOOL  ; 読出し中
W312.01 BOOL  ; 読出し完
W312.02 BOOL  ; ﾃﾞｰﾀ無読出中止
W312.03 BOOL  ; 出力ｴﾘｱ空2
W312.04 BOOL  ; 出力ｴﾘｱ空3
W312.05 BOOL  ; 出力ｴﾘｱ空4
W312.06 BOOL  ; 出力ｴﾘｱ空
W312.07 BOOL  ; chk1
W312.08 BOOL  ; chk2
W312.09 BOOL  ; chk3
W312.10 BOOL  ; chk4
W312.11 BOOL  ; chk5
W312.12 BOOL  ; chk6
W312.13 BOOL  ; chk7
W312.14 BOOL  ; chk8
W313.00 BOOL  ; Dエリアクリア開始
W313.01 BOOL  ; Dエリアクリア完
W313.02 BOOL  ; ﾃﾞｰﾀｴﾘｱｸﾘｱ_ﾄﾘｶﾞ
W313.03 BOOL  ; PC_First_cycle
W313.04 BOOL  ; PC_Starc_Clear
W313.05 BOOL  ; tchk1
W313.06 BOOL  ; tchk2
W313.07 BOOL  ; tchk3
W313.08 BOOL  ; tchk4
W313.09 BOOL  ; tchk5
W313.10 BOOL  ; TMP有効ﾃﾞｰﾀ無
W314.00 BOOL  ; PV_result
W314.01 BOOL  ; DV_result
W314.02 BOOL  ; TSO_result
W314.03 BOOL  ; NC_result
W314.04 BOOL  ; NO_result
W314.05 BOOL  ; CG_result
W314.06 BOOL  ; CG_result
W319.00 BOOL  ; 入力ｴﾘｱ無
W319.01 BOOL  ; 入力ｴﾘｱ有
W319.02 BOOL  ; 出力ｴﾘｱ無
W319.03 BOOL  ; 出力ｴﾘｱ有
W321.00 BOOL  ; 読み込み中
W321.01 BOOL  ; 読込み完
W350.00 BOOL  ; Ready_RT_hold
W350.01 BOOL  ; Ready_MVD_hold
W360.00 BOOL  ; 取出hold
W400.00 BOOL  ; -
W400.01 BOOL  ; -
W400.03 BOOL  ; -
W400.04 BOOL  ; -
W401.00 BOOL  ; -
W401.01 BOOL  ; -
W401.02 BOOL  ; -
W401.03 BOOL  ; -
W401.04 BOOL  ; -
W401.05 BOOL  ; -
W401.06 BOOL  ; -
W402.00 BOOL  ; -
W402.01 BOOL  ; -
W402.02 BOOL  ; -
W402.03 BOOL  ; -
W402.04 BOOL  ; -
W402.05 BOOL  ; -
W402.06 BOOL  ; -
W402.07 BOOL  ; -
W402.08 BOOL  ; -
W402.09 BOOL  ; -
W402.10 BOOL  ; -
W403.00 BOOL  ; -
W500.00 BOOL  ; -
W500.01 BOOL  ; -
W500.02 BOOL  ; -
W500.03 BOOL  ; -
W500.04 BOOL  ; -
W500.05 BOOL  ; -
W500.06 BOOL  ; -
W500.07 BOOL  ; -
W500.08 BOOL  ; -
W500.09 BOOL  ; -
W500.10 BOOL  ; -
W500.11 BOOL  ; -
W500.12 BOOL  ; -
W500.13 BOOL  ; -
W500.14 BOOL  ; -
W501.00 BOOL  ; -
W501.01 BOOL  ; -
W501.02 BOOL  ; -
W502.00 BOOL  ; -
W502.01 BOOL  ; -
W503.00 BOOL  ; 時刻設定開始
W503.01 BOOL  ; 時刻設定中
W503.02 BOOL  ; 時刻変更終了
W503.03 BOOL  ; 時刻設定完了
W504.00 BOOL  ; -
W504.01 BOOL  ; -
W504.02 BOOL  ; -
W504.03 BOOL  ; -
W504.04 BOOL  ; -
W504.05 BOOL  ; -
W505.00 BOOL  ; -
W505.01 BOOL  ; -
W505.02 BOOL  ; -
W511.00 BOOL  ; -
W511.01 BOOL  ; -
W511.02 BOOL  ; -
W5.02 BOOL  ; LCAM_TRIG
W5.03 BOOL  ; LCAM_BUSY
W5.04 BOOL  ; LCAM_RESULT
W60.01 BOOL  ; lt_cam_trigger_hold
W6.00 BOOL  ; データ読込開始
W6.04 BOOL  ; palette_set_ok
W99.15 BOOL  ; DebugMode

## Program ﾃﾞｰﾀ収集PLCﾌﾟﾛｸﾞﾗﾑ (cyclic task 1)
Local symbols
D13500D13501 INT
l CHANNEL  ; CH1PV

### Section 初期設定

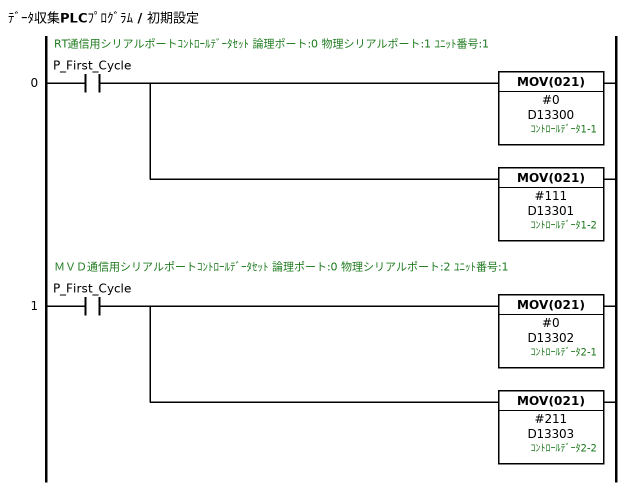
; rung 0: RT通信用シリアルポートｺﾝﾄﾛｰﾙﾃﾞｰﾀｾｯﾄ 論理ポート:0 物理シリアルポート:1 ﾕﾆｯﾄ番号:1
LD P_First_Cycle
MOV(021) #0 D13300  ; ｺﾝﾄﾛｰﾙﾃﾞｰﾀ1-1
MOV(021) #111 D13301  ; ｺﾝﾄﾛｰﾙﾃﾞｰﾀ1-2
; rung 1: ＭＶＤ通信用シリアルポートｺﾝﾄﾛｰﾙﾃﾞｰﾀｾｯﾄ 論理ポート:0 物理シリアルポート:2 ﾕﾆｯﾄ番号:1
LD P_First_Cycle
MOV(021) #0 D13302  ; ｺﾝﾄﾛｰﾙﾃﾞｰﾀ2-1
MOV(021) #211 D13303  ; ｺﾝﾄﾛｰﾙﾃﾞｰﾀ2-2

### Section PC･搬送PLC制御通信

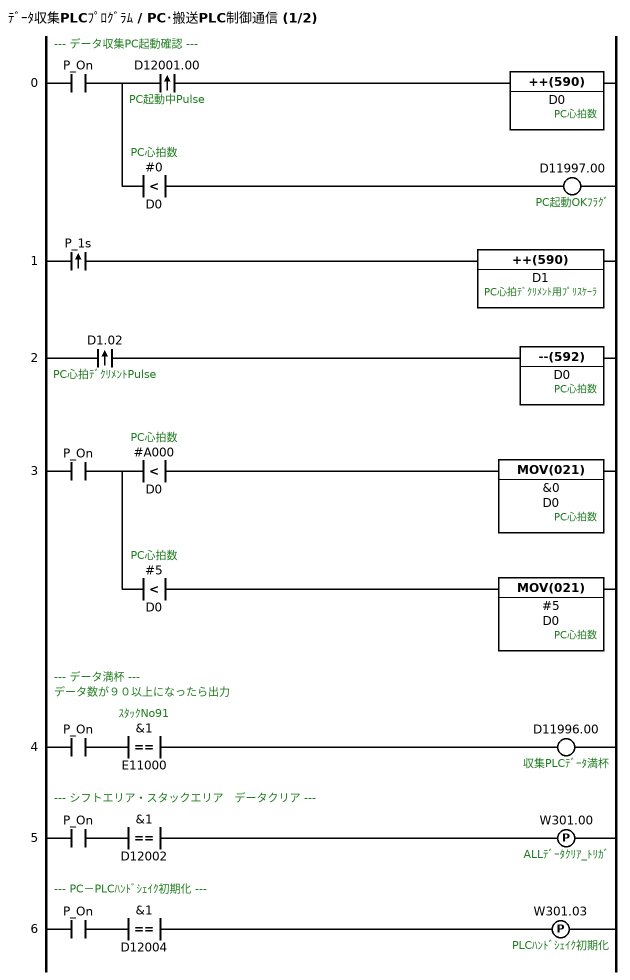
; rung 0: --- データ収集PC起動確認 ---
LD P_On
OUT TR0
@AND D12001.00  ; PC起動中Pulse
++(590) D0  ; PC心拍数
LD TR0
AND<(310) #0 D0  ; PC心拍数
OUT D11997.00  ; PC起動OKﾌﾗｸﾞ
; rung 1
@LD P_1s
++(590) D1  ; PC心拍ﾃﾞｸﾘﾒﾝﾄ用ﾌﾟﾘｽｹｰﾗ
; rung 2
@LD D1.02  ; PC心拍ﾃﾞｸﾘﾒﾝﾄPulse
--(592) D0  ; PC心拍数
; rung 3
LD P_On
OUT TR0
AND<(310) #A000 D0  ; PC心拍数
MOV(021) &0 D0  ; PC心拍数
LD TR0
AND<(310) #5 D0  ; PC心拍数
MOV(021) #5 D0  ; PC心拍数
; rung 4: --- データ満杯 --- / データ数が９０以上になったら出力
LD P_On
AND=(300) &1 E11000  ; ｽﾀｯｸNo91
OUT D11996.00  ; 収集PLCﾃﾞｰﾀ満杯
; rung 5: --- シフトエリア・スタックエリア　データクリア ---
LD P_On
AND=(300) &1 D12002
DIFU(013) W301.00  ; ALLﾃﾞｰﾀｸﾘｱ_ﾄﾘｶﾞ
; rung 6: --- PC－PLCﾊﾝﾄﾞｼｪｲｸ初期化 ---
LD P_On
AND=(300) &1 D12004
DIFU(013) W301.03  ; PLCﾊﾝﾄﾞｼｪｲｸ初期化

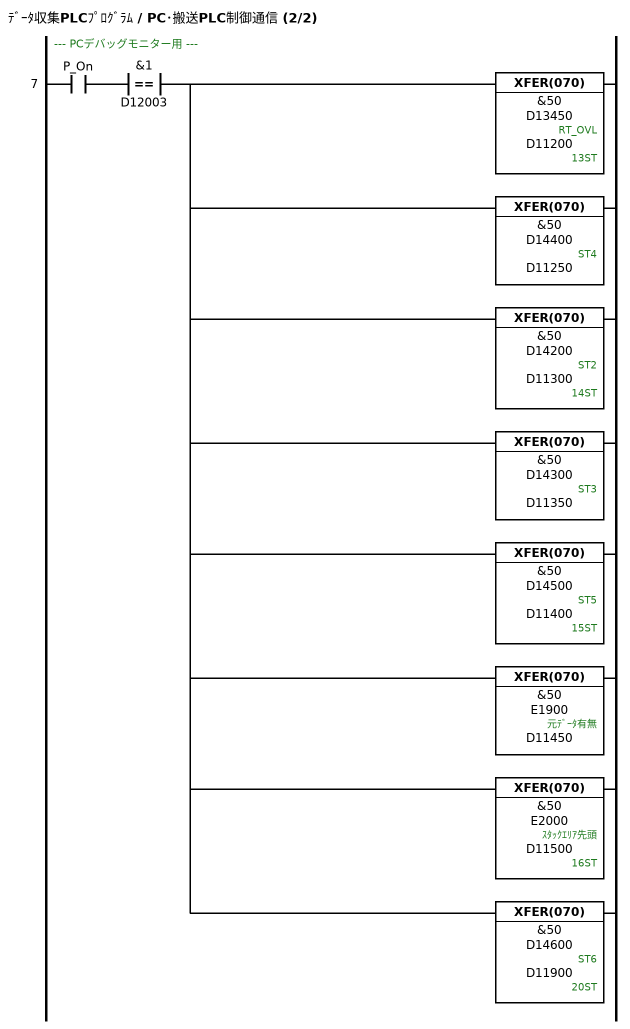
; rung 7: --- PCデバッグモニター用 ---
LD P_On
AND=(300) &1 D12003
XFER(070) &50 D13450 D11200  ; RT_OVL, 13ST
XFER(070) &50 D14400 D11250  ; ST4
XFER(070) &50 D14200 D11300  ; ST2, 14ST
XFER(070) &50 D14300 D11350  ; ST3
XFER(070) &50 D14500 D11400  ; ST5, 15ST
XFER(070) &50 E1900 D11450  ; 元ﾃﾞｰﾀ有無
XFER(070) &50 E2000 D11500  ; ｽﾀｯｸｴﾘｱ先頭, 16ST
XFER(070) &50 D14600 D11900  ; ST6, 20ST

### Section Ch1特性検査Unit通信開始

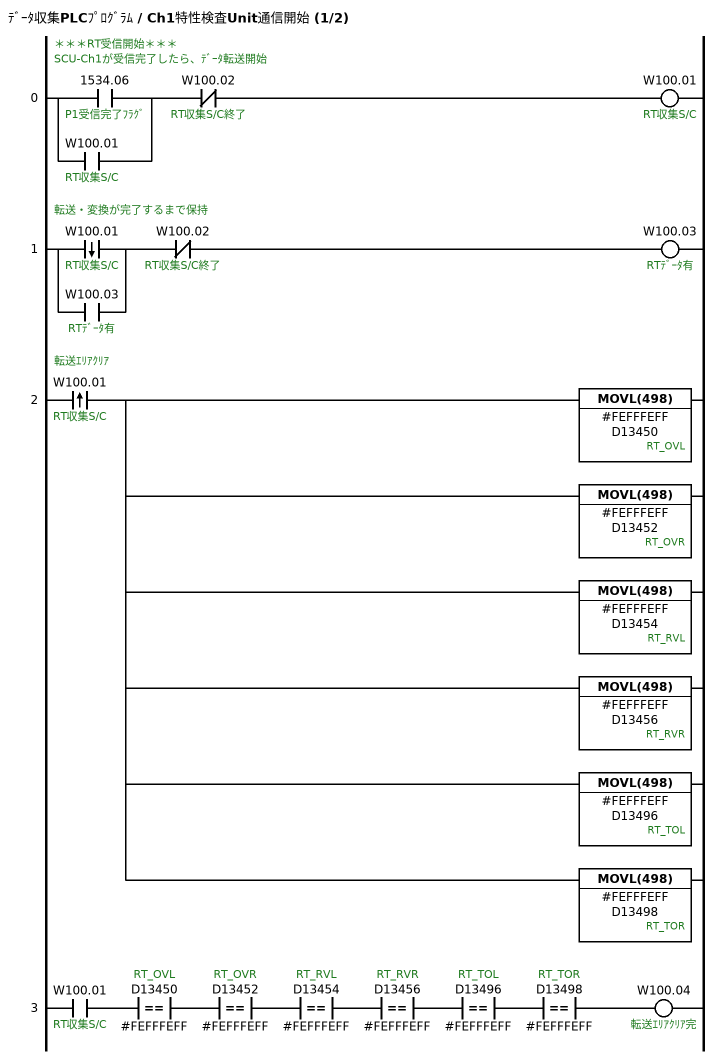
; rung 0: ＊＊＊RT受信開始＊＊＊ / SCU-Ch1が受信完了したら、ﾃﾞｰﾀ転送開始
LD 1534.06  ; P1受信完了ﾌﾗｸﾞ
OR W100.01  ; RT収集S/C
ANDNOT W100.02  ; RT収集S/C終了
OUT W100.01  ; RT収集S/C
; rung 1: 転送・変換が完了するまで保持
%LD W100.01  ; RT収集S/C
OR W100.03  ; RTﾃﾞｰﾀ有
ANDNOT W100.02  ; RT収集S/C終了
OUT W100.03  ; RTﾃﾞｰﾀ有
; rung 2: 転送ｴﾘｱｸﾘｱ
@LD W100.01  ; RT収集S/C
MOVL(498) #FEFFFEFF D13450  ; RT_OVL
MOVL(498) #FEFFFEFF D13452  ; RT_OVR
MOVL(498) #FEFFFEFF D13454  ; RT_RVL
MOVL(498) #FEFFFEFF D13456  ; RT_RVR
MOVL(498) #FEFFFEFF D13496  ; RT_TOL
MOVL(498) #FEFFFEFF D13498  ; RT_TOR
; rung 3
LD W100.01  ; RT収集S/C
AND=L(301) D13450 #FEFFFEFF  ; RT_OVL
AND=L(301) D13452 #FEFFFEFF  ; RT_OVR
AND=L(301) D13454 #FEFFFEFF  ; RT_RVL
AND=L(301) D13456 #FEFFFEFF  ; RT_RVR
AND=L(301) D13496 #FEFFFEFF  ; RT_TOL
AND=L(301) D13498 #FEFFFEFF  ; RT_TOR
OUT W100.04  ; 転送ｴﾘｱｸﾘｱ完

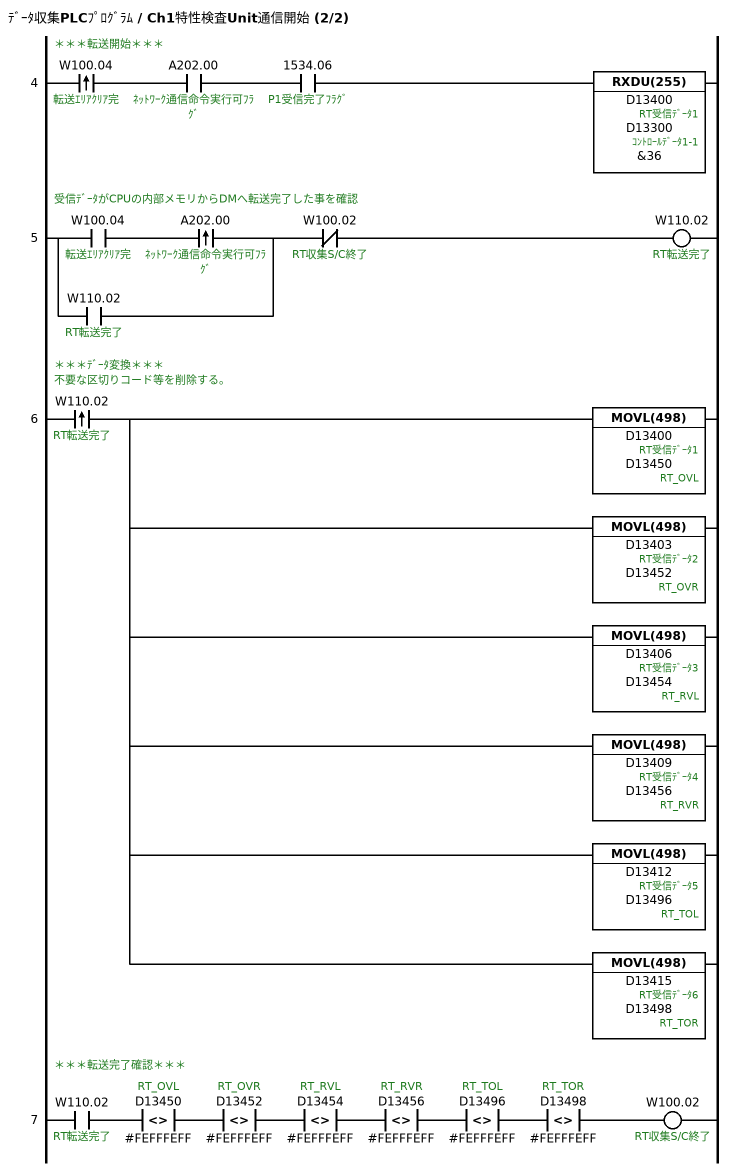
; rung 4: ＊＊＊転送開始＊＊＊
@LD W100.04  ; 転送ｴﾘｱｸﾘｱ完
AND A202.00  ; ﾈｯﾄﾜｰｸ通信命令実行可ﾌﾗｸﾞ
AND 1534.06  ; P1受信完了ﾌﾗｸﾞ
RXDU(255) D13400 D13300 &36  ; RT受信ﾃﾞｰﾀ1, ｺﾝﾄﾛｰﾙﾃﾞｰﾀ1-1
; rung 5: 受信ﾃﾞｰﾀがCPUの内部メモリからDMへ転送完了した事を確認
LD W100.04  ; 転送ｴﾘｱｸﾘｱ完
@AND A202.00  ; ﾈｯﾄﾜｰｸ通信命令実行可ﾌﾗｸﾞ
OR W110.02  ; RT転送完了
ANDNOT W100.02  ; RT収集S/C終了
OUT W110.02  ; RT転送完了
; rung 6: ＊＊＊ﾃﾞｰﾀ変換＊＊＊ / 不要な区切りコード等を削除する。
@LD W110.02  ; RT転送完了
MOVL(498) D13400 D13450  ; RT受信ﾃﾞｰﾀ1, RT_OVL
MOVL(498) D13403 D13452  ; RT受信ﾃﾞｰﾀ2, RT_OVR
MOVL(498) D13406 D13454  ; RT受信ﾃﾞｰﾀ3, RT_RVL
MOVL(498) D13409 D13456  ; RT受信ﾃﾞｰﾀ4, RT_RVR
MOVL(498) D13412 D13496  ; RT受信ﾃﾞｰﾀ5, RT_TOL
MOVL(498) D13415 D13498  ; RT受信ﾃﾞｰﾀ6, RT_TOR
; rung 7: ＊＊＊転送完了確認＊＊＊
LD W110.02  ; RT転送完了
AND<>L(306) D13450 #FEFFFEFF  ; RT_OVL
AND<>L(306) D13452 #FEFFFEFF  ; RT_OVR
AND<>L(306) D13454 #FEFFFEFF  ; RT_RVL
AND<>L(306) D13456 #FEFFFEFF  ; RT_RVR
AND<>L(306) D13496 #FEFFFEFF  ; RT_TOL
AND<>L(306) D13498 #FEFFFEFF  ; RT_TOR
OUT W100.02  ; RT収集S/C終了

### Section Ch2CP検査Unit通信開始

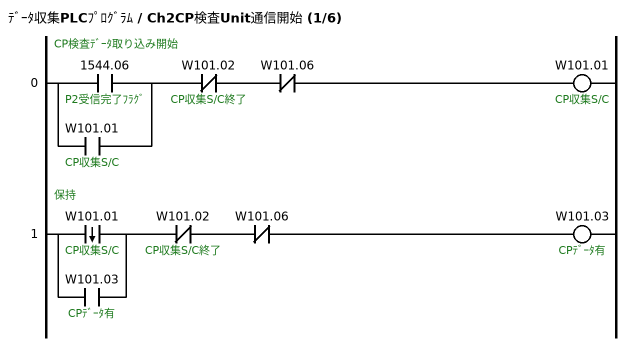
; rung 0: CP検査ﾃﾞｰﾀ取り込み開始
LD 1544.06  ; P2受信完了ﾌﾗｸﾞ
OR W101.01  ; CP収集S/C
ANDNOT W101.02  ; CP収集S/C終了
ANDNOT W101.06
OUT W101.01  ; CP収集S/C
; rung 1: 保持
%LD W101.01  ; CP収集S/C
OR W101.03  ; CPﾃﾞｰﾀ有
ANDNOT W101.02  ; CP収集S/C終了
ANDNOT W101.06
OUT W101.03  ; CPﾃﾞｰﾀ有

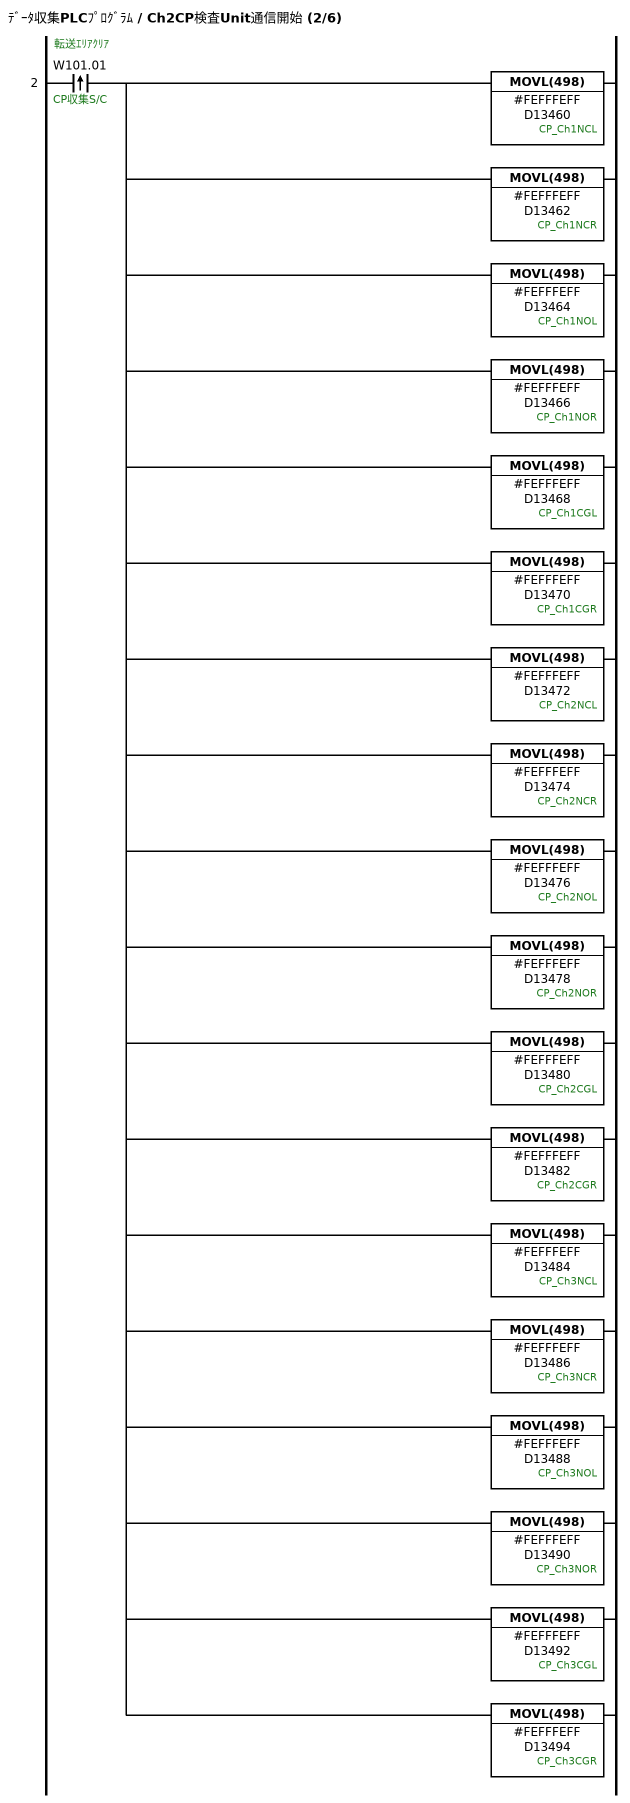
; rung 2: 転送ｴﾘｱｸﾘｱ
@LD W101.01  ; CP収集S/C
MOVL(498) #FEFFFEFF D13460  ; CP_Ch1NCL
MOVL(498) #FEFFFEFF D13462  ; CP_Ch1NCR
MOVL(498) #FEFFFEFF D13464  ; CP_Ch1NOL
MOVL(498) #FEFFFEFF D13466  ; CP_Ch1NOR
MOVL(498) #FEFFFEFF D13468  ; CP_Ch1CGL
MOVL(498) #FEFFFEFF D13470  ; CP_Ch1CGR
MOVL(498) #FEFFFEFF D13472  ; CP_Ch2NCL
MOVL(498) #FEFFFEFF D13474  ; CP_Ch2NCR
MOVL(498) #FEFFFEFF D13476  ; CP_Ch2NOL
MOVL(498) #FEFFFEFF D13478  ; CP_Ch2NOR
MOVL(498) #FEFFFEFF D13480  ; CP_Ch2CGL
MOVL(498) #FEFFFEFF D13482  ; CP_Ch2CGR
MOVL(498) #FEFFFEFF D13484  ; CP_Ch3NCL
MOVL(498) #FEFFFEFF D13486  ; CP_Ch3NCR
MOVL(498) #FEFFFEFF D13488  ; CP_Ch3NOL
MOVL(498) #FEFFFEFF D13490  ; CP_Ch3NOR
MOVL(498) #FEFFFEFF D13492  ; CP_Ch3CGL
MOVL(498) #FEFFFEFF D13494  ; CP_Ch3CGR

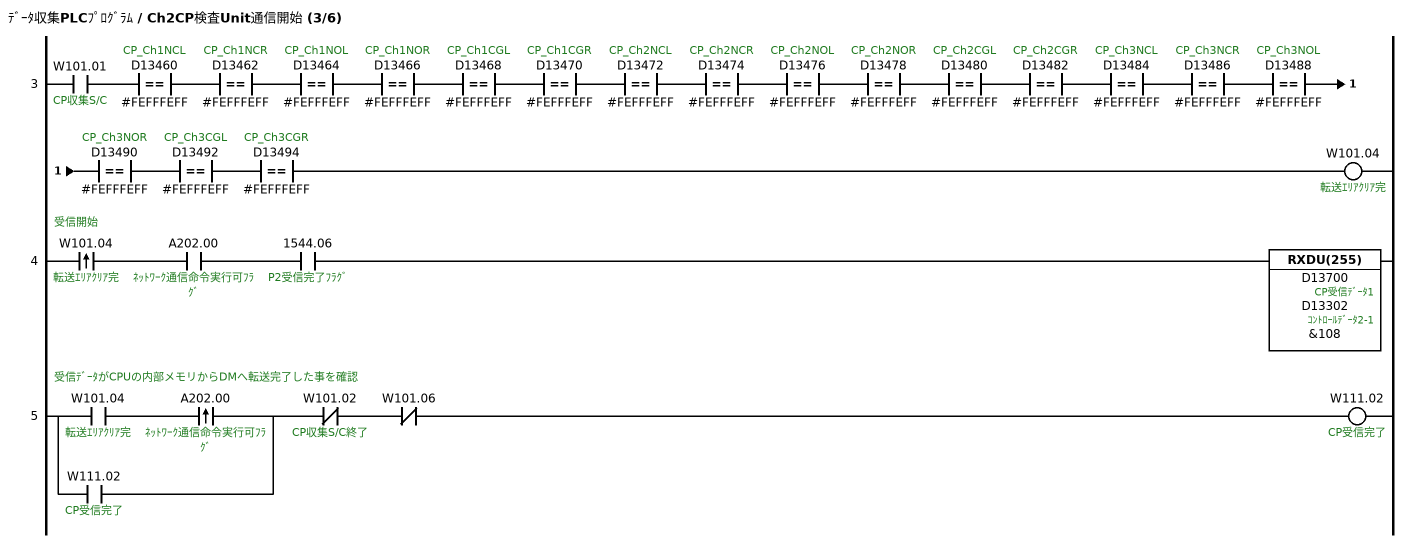
; rung 3
LD W101.01  ; CP収集S/C
AND=L(301) D13460 #FEFFFEFF  ; CP_Ch1NCL
AND=L(301) D13462 #FEFFFEFF  ; CP_Ch1NCR
AND=L(301) D13464 #FEFFFEFF  ; CP_Ch1NOL
AND=L(301) D13466 #FEFFFEFF  ; CP_Ch1NOR
AND=L(301) D13468 #FEFFFEFF  ; CP_Ch1CGL
AND=L(301) D13470 #FEFFFEFF  ; CP_Ch1CGR
AND=L(301) D13472 #FEFFFEFF  ; CP_Ch2NCL
AND=L(301) D13474 #FEFFFEFF  ; CP_Ch2NCR
AND=L(301) D13476 #FEFFFEFF  ; CP_Ch2NOL
AND=L(301) D13478 #FEFFFEFF  ; CP_Ch2NOR
AND=L(301) D13480 #FEFFFEFF  ; CP_Ch2CGL
AND=L(301) D13482 #FEFFFEFF  ; CP_Ch2CGR
AND=L(301) D13484 #FEFFFEFF  ; CP_Ch3NCL
AND=L(301) D13486 #FEFFFEFF  ; CP_Ch3NCR
AND=L(301) D13488 #FEFFFEFF  ; CP_Ch3NOL
AND=L(301) D13490 #FEFFFEFF  ; CP_Ch3NOR
AND=L(301) D13492 #FEFFFEFF  ; CP_Ch3CGL
AND=L(301) D13494 #FEFFFEFF  ; CP_Ch3CGR
OUT W101.04  ; 転送ｴﾘｱｸﾘｱ完
; rung 4: 受信開始
@LD W101.04  ; 転送ｴﾘｱｸﾘｱ完
AND A202.00  ; ﾈｯﾄﾜｰｸ通信命令実行可ﾌﾗｸﾞ
AND 1544.06  ; P2受信完了ﾌﾗｸﾞ
RXDU(255) D13700 D13302 &108  ; CP受信ﾃﾞｰﾀ1, ｺﾝﾄﾛｰﾙﾃﾞｰﾀ2-1
; rung 5: 受信ﾃﾞｰﾀがCPUの内部メモリからDMへ転送完了した事を確認
LD W101.04  ; 転送ｴﾘｱｸﾘｱ完
@AND A202.00  ; ﾈｯﾄﾜｰｸ通信命令実行可ﾌﾗｸﾞ
OR W111.02  ; CP受信完了
ANDNOT W101.02  ; CP収集S/C終了
ANDNOT W101.06
OUT W111.02  ; CP受信完了

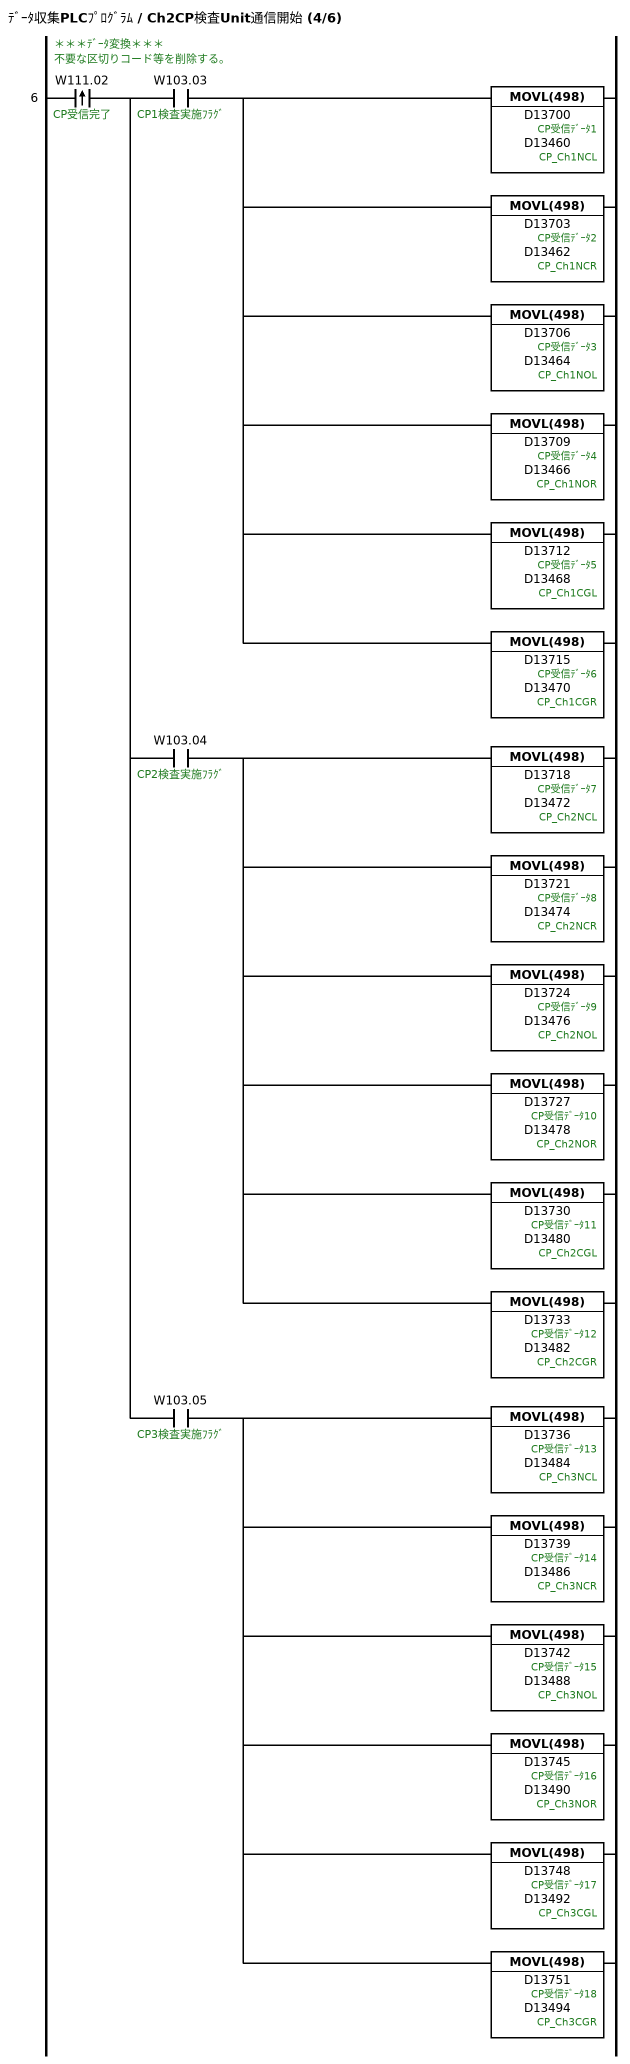
; rung 6: ＊＊＊ﾃﾞｰﾀ変換＊＊＊ / 不要な区切りコード等を削除する。
@LD W111.02  ; CP受信完了
OUT TR0
AND W103.03  ; CP1検査実施ﾌﾗｸﾞ
MOVL(498) D13700 D13460  ; CP受信ﾃﾞｰﾀ1, CP_Ch1NCL
MOVL(498) D13703 D13462  ; CP受信ﾃﾞｰﾀ2, CP_Ch1NCR
MOVL(498) D13706 D13464  ; CP受信ﾃﾞｰﾀ3, CP_Ch1NOL
MOVL(498) D13709 D13466  ; CP受信ﾃﾞｰﾀ4, CP_Ch1NOR
MOVL(498) D13712 D13468  ; CP受信ﾃﾞｰﾀ5, CP_Ch1CGL
MOVL(498) D13715 D13470  ; CP受信ﾃﾞｰﾀ6, CP_Ch1CGR
LD TR0
AND W103.04  ; CP2検査実施ﾌﾗｸﾞ
MOVL(498) D13718 D13472  ; CP受信ﾃﾞｰﾀ7, CP_Ch2NCL
MOVL(498) D13721 D13474  ; CP受信ﾃﾞｰﾀ8, CP_Ch2NCR
MOVL(498) D13724 D13476  ; CP受信ﾃﾞｰﾀ9, CP_Ch2NOL
MOVL(498) D13727 D13478  ; CP受信ﾃﾞｰﾀ10, CP_Ch2NOR
MOVL(498) D13730 D13480  ; CP受信ﾃﾞｰﾀ11, CP_Ch2CGL
MOVL(498) D13733 D13482  ; CP受信ﾃﾞｰﾀ12, CP_Ch2CGR
LD TR0
AND W103.05  ; CP3検査実施ﾌﾗｸﾞ
MOVL(498) D13736 D13484  ; CP受信ﾃﾞｰﾀ13, CP_Ch3NCL
MOVL(498) D13739 D13486  ; CP受信ﾃﾞｰﾀ14, CP_Ch3NCR
MOVL(498) D13742 D13488  ; CP受信ﾃﾞｰﾀ15, CP_Ch3NOL
MOVL(498) D13745 D13490  ; CP受信ﾃﾞｰﾀ16, CP_Ch3NOR
MOVL(498) D13748 D13492  ; CP受信ﾃﾞｰﾀ17, CP_Ch3CGL
MOVL(498) D13751 D13494  ; CP受信ﾃﾞｰﾀ18, CP_Ch3CGR

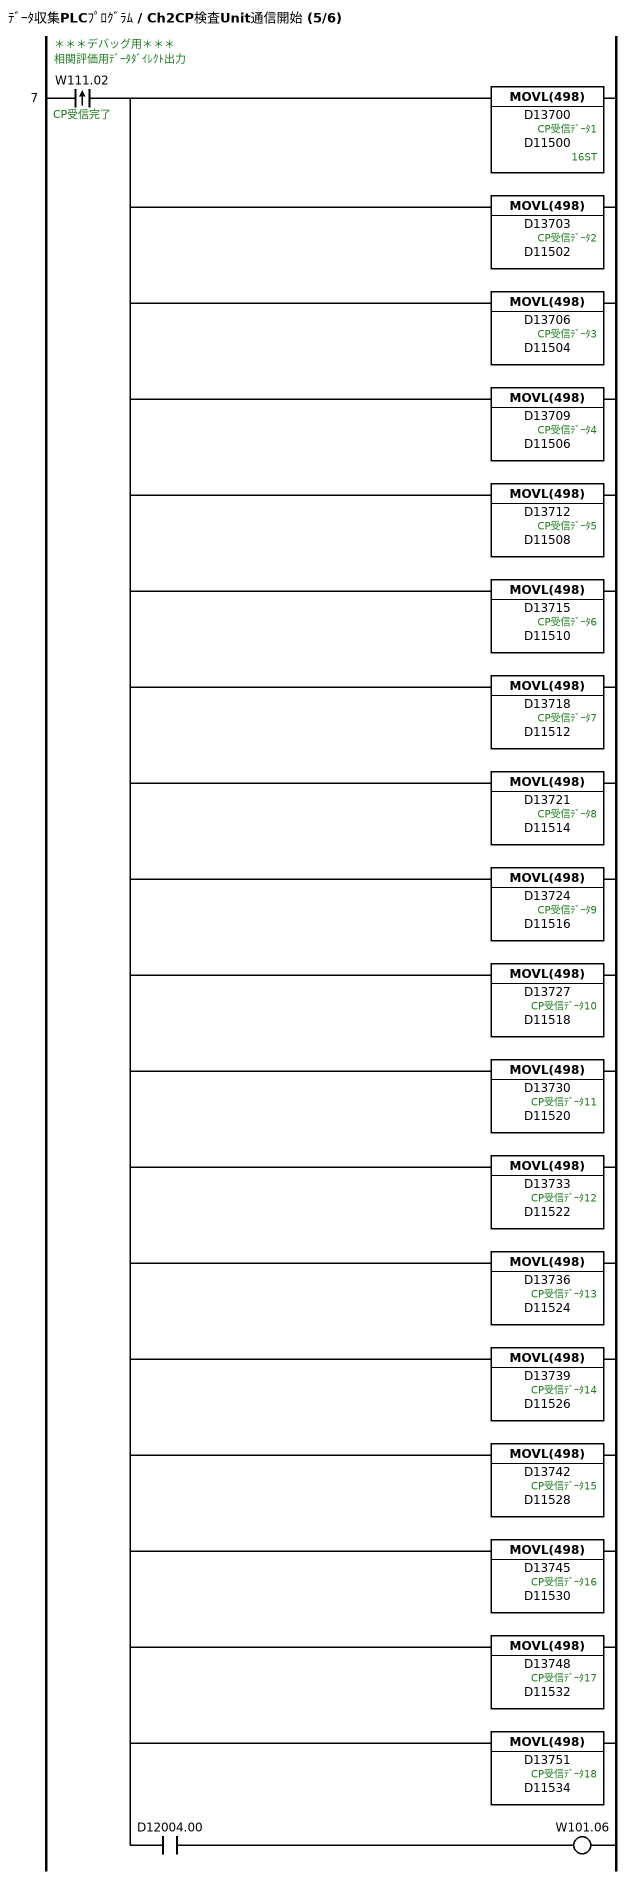
; rung 7: ＊＊＊デバッグ用＊＊＊ / 相関評価用ﾃﾞｰﾀﾀﾞｲﾚｸﾄ出力
@LD W111.02  ; CP受信完了
MOVL(498) D13700 D11500  ; CP受信ﾃﾞｰﾀ1, 16ST
MOVL(498) D13703 D11502  ; CP受信ﾃﾞｰﾀ2
MOVL(498) D13706 D11504  ; CP受信ﾃﾞｰﾀ3
MOVL(498) D13709 D11506  ; CP受信ﾃﾞｰﾀ4
MOVL(498) D13712 D11508  ; CP受信ﾃﾞｰﾀ5
MOVL(498) D13715 D11510  ; CP受信ﾃﾞｰﾀ6
MOVL(498) D13718 D11512  ; CP受信ﾃﾞｰﾀ7
MOVL(498) D13721 D11514  ; CP受信ﾃﾞｰﾀ8
MOVL(498) D13724 D11516  ; CP受信ﾃﾞｰﾀ9
MOVL(498) D13727 D11518  ; CP受信ﾃﾞｰﾀ10
MOVL(498) D13730 D11520  ; CP受信ﾃﾞｰﾀ11
MOVL(498) D13733 D11522  ; CP受信ﾃﾞｰﾀ12
MOVL(498) D13736 D11524  ; CP受信ﾃﾞｰﾀ13
MOVL(498) D13739 D11526  ; CP受信ﾃﾞｰﾀ14
MOVL(498) D13742 D11528  ; CP受信ﾃﾞｰﾀ15
MOVL(498) D13745 D11530  ; CP受信ﾃﾞｰﾀ16
MOVL(498) D13748 D11532  ; CP受信ﾃﾞｰﾀ17
MOVL(498) D13751 D11534  ; CP受信ﾃﾞｰﾀ18
AND D12004.00
OUT W101.06

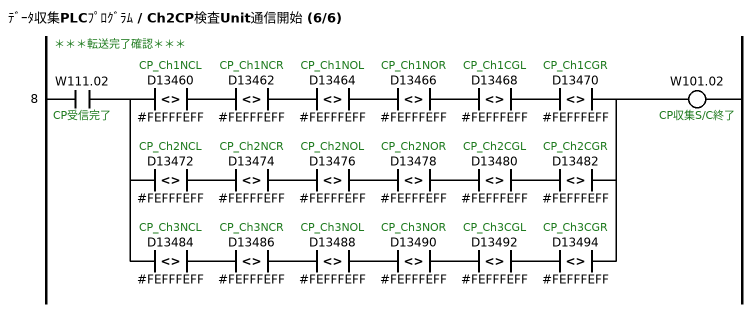
; rung 8: ＊＊＊転送完了確認＊＊＊
LD W111.02  ; CP受信完了
LD<>L(306) D13460 #FEFFFEFF  ; CP_Ch1NCL
AND<>L(306) D13462 #FEFFFEFF  ; CP_Ch1NCR
AND<>L(306) D13464 #FEFFFEFF  ; CP_Ch1NOL
AND<>L(306) D13466 #FEFFFEFF  ; CP_Ch1NOR
AND<>L(306) D13468 #FEFFFEFF  ; CP_Ch1CGL
AND<>L(306) D13470 #FEFFFEFF  ; CP_Ch1CGR
LD<>L(306) D13472 #FEFFFEFF  ; CP_Ch2NCL
AND<>L(306) D13474 #FEFFFEFF  ; CP_Ch2NCR
AND<>L(306) D13476 #FEFFFEFF  ; CP_Ch2NOL
AND<>L(306) D13478 #FEFFFEFF  ; CP_Ch2NOR
AND<>L(306) D13480 #FEFFFEFF  ; CP_Ch2CGL
AND<>L(306) D13482 #FEFFFEFF  ; CP_Ch2CGR
ORLD
LD<>L(306) D13484 #FEFFFEFF  ; CP_Ch3NCL
AND<>L(306) D13486 #FEFFFEFF  ; CP_Ch3NCR
AND<>L(306) D13488 #FEFFFEFF  ; CP_Ch3NOL
AND<>L(306) D13490 #FEFFFEFF  ; CP_Ch3NOR
AND<>L(306) D13492 #FEFFFEFF  ; CP_Ch3CGL
AND<>L(306) D13494 #FEFFFEFF  ; CP_Ch3CGR
ORLD
ANDLD
OUT W101.02  ; CP収集S/C終了

### Section ｼﾌﾄｴﾘｱ_ﾃﾞｰﾀ書込み･ｼﾌﾄ

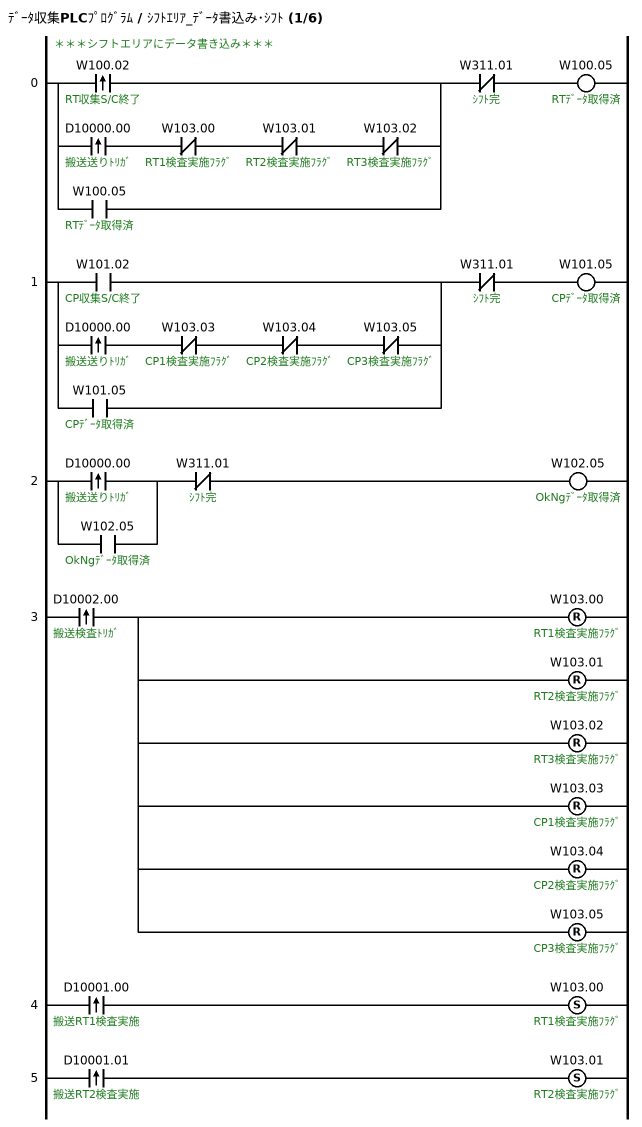
; rung 0: ＊＊＊シフトエリアにデータ書き込み＊＊＊
@LD W100.02  ; RT収集S/C終了
@LD D10000.00  ; 搬送送りﾄﾘｶﾞ
ANDNOT W103.00  ; RT1検査実施ﾌﾗｸﾞ
ANDNOT W103.01  ; RT2検査実施ﾌﾗｸﾞ
ANDNOT W103.02  ; RT3検査実施ﾌﾗｸﾞ
ORLD
OR W100.05  ; RTﾃﾞｰﾀ取得済
ANDNOT W311.01  ; ｼﾌﾄ完
OUT W100.05  ; RTﾃﾞｰﾀ取得済
; rung 1
LD W101.02  ; CP収集S/C終了
@LD D10000.00  ; 搬送送りﾄﾘｶﾞ
ANDNOT W103.03  ; CP1検査実施ﾌﾗｸﾞ
ANDNOT W103.04  ; CP2検査実施ﾌﾗｸﾞ
ANDNOT W103.05  ; CP3検査実施ﾌﾗｸﾞ
ORLD
OR W101.05  ; CPﾃﾞｰﾀ取得済
ANDNOT W311.01  ; ｼﾌﾄ完
OUT W101.05  ; CPﾃﾞｰﾀ取得済
; rung 2
@LD D10000.00  ; 搬送送りﾄﾘｶﾞ
OR W102.05  ; OkNgﾃﾞｰﾀ取得済
ANDNOT W311.01  ; ｼﾌﾄ完
OUT W102.05  ; OkNgﾃﾞｰﾀ取得済
; rung 3
@LD D10002.00  ; 搬送検査ﾄﾘｶﾞ
RSET W103.00  ; RT1検査実施ﾌﾗｸﾞ
RSET W103.01  ; RT2検査実施ﾌﾗｸﾞ
RSET W103.02  ; RT3検査実施ﾌﾗｸﾞ
RSET W103.03  ; CP1検査実施ﾌﾗｸﾞ
RSET W103.04  ; CP2検査実施ﾌﾗｸﾞ
RSET W103.05  ; CP3検査実施ﾌﾗｸﾞ
; rung 4
@LD D10001.00  ; 搬送RT1検査実施
SET W103.00  ; RT1検査実施ﾌﾗｸﾞ
; rung 5
@LD D10001.01  ; 搬送RT2検査実施
SET W103.01  ; RT2検査実施ﾌﾗｸﾞ

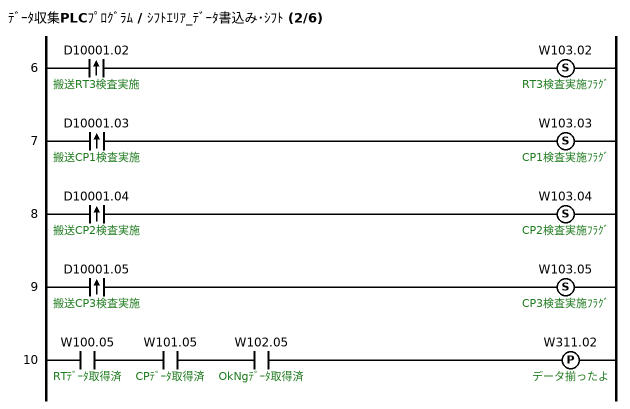
; rung 6
@LD D10001.02  ; 搬送RT3検査実施
SET W103.02  ; RT3検査実施ﾌﾗｸﾞ
; rung 7
@LD D10001.03  ; 搬送CP1検査実施
SET W103.03  ; CP1検査実施ﾌﾗｸﾞ
; rung 8
@LD D10001.04  ; 搬送CP2検査実施
SET W103.04  ; CP2検査実施ﾌﾗｸﾞ
; rung 9
@LD D10001.05  ; 搬送CP3検査実施
SET W103.05  ; CP3検査実施ﾌﾗｸﾞ
; rung 10
LD W100.05  ; RTﾃﾞｰﾀ取得済
AND W101.05  ; CPﾃﾞｰﾀ取得済
AND W102.05  ; OkNgﾃﾞｰﾀ取得済
DIFU(013) W311.02  ; データ揃ったよ

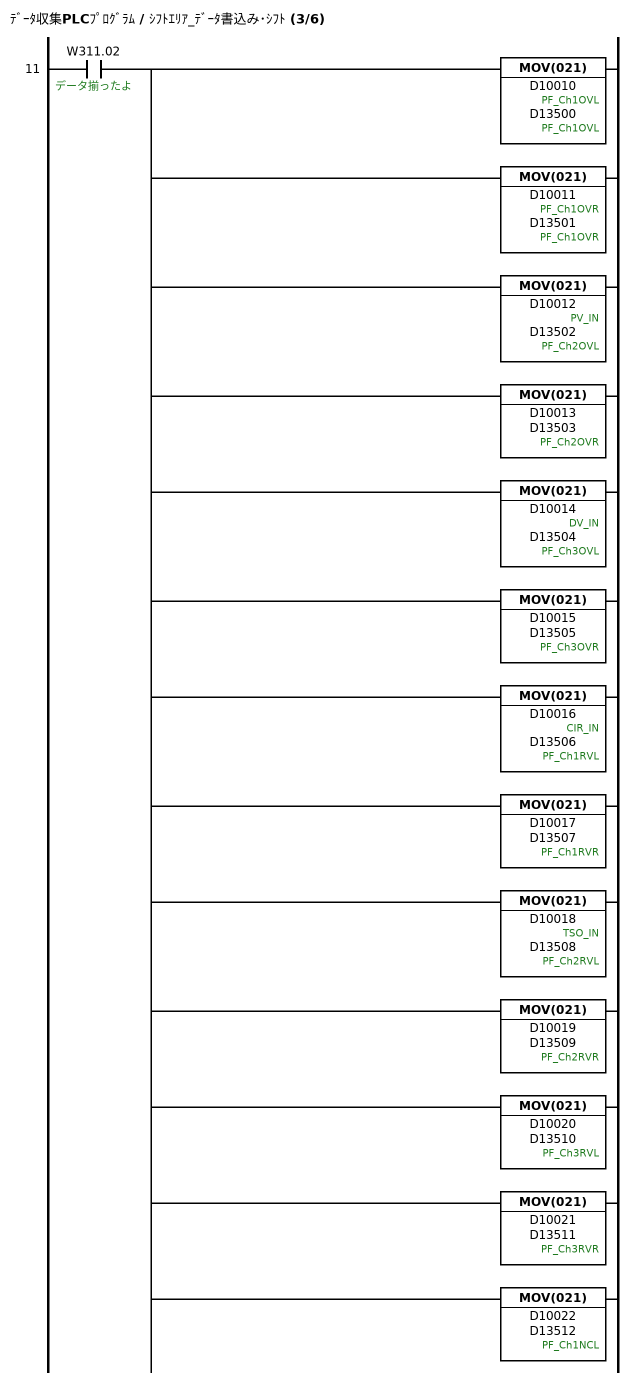

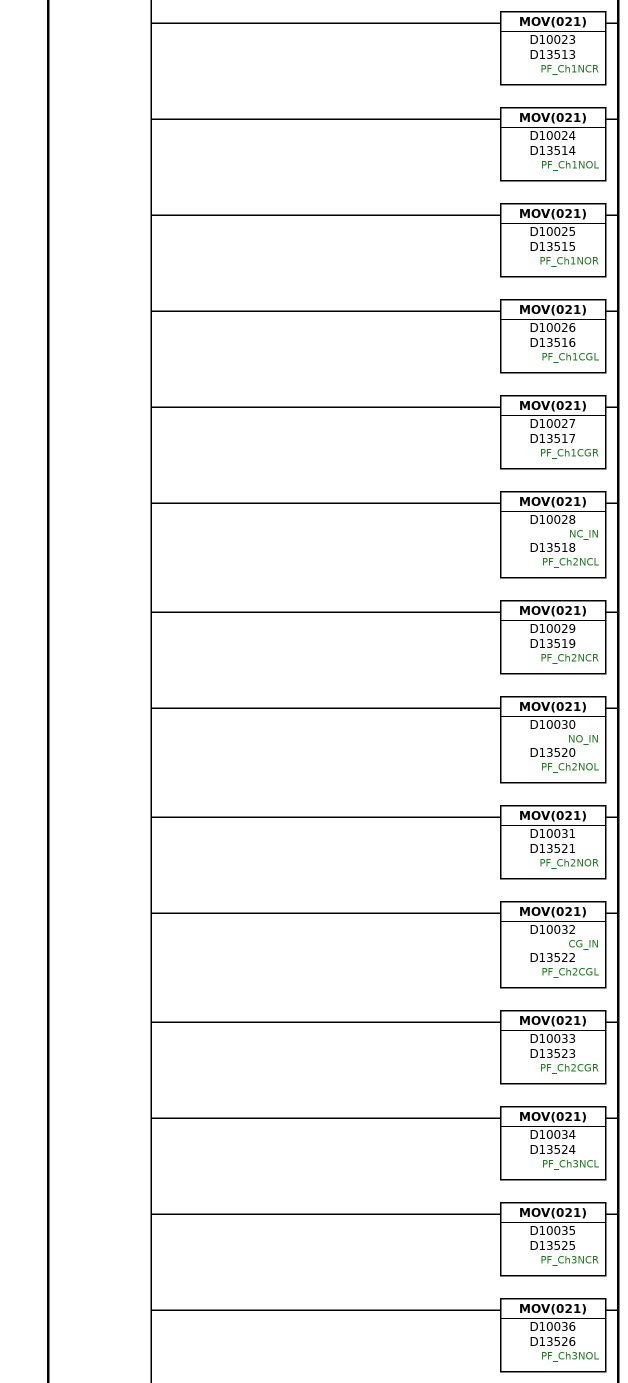

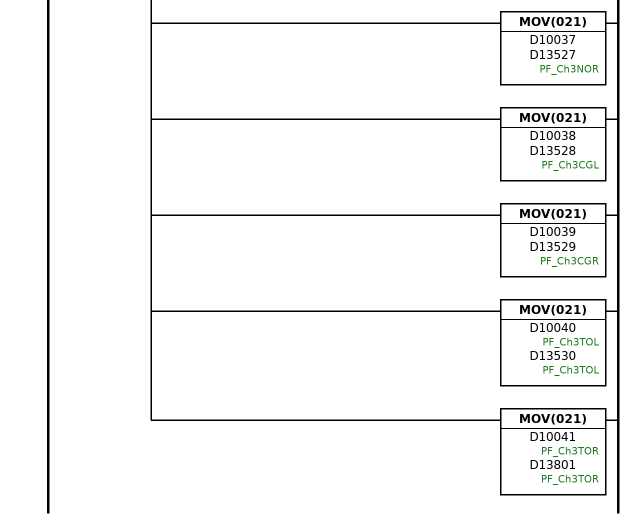
; rung 11
LD W311.02  ; データ揃ったよ
MOV(021) D10010 D13500  ; PF_Ch1OVL
MOV(021) D10011 D13501  ; PF_Ch1OVR
MOV(021) D10012 D13502  ; PV_IN, PF_Ch2OVL
MOV(021) D10013 D13503  ; PF_Ch2OVR
MOV(021) D10014 D13504  ; DV_IN, PF_Ch3OVL
MOV(021) D10015 D13505  ; PF_Ch3OVR
MOV(021) D10016 D13506  ; CIR_IN, PF_Ch1RVL
MOV(021) D10017 D13507  ; PF_Ch1RVR
MOV(021) D10018 D13508  ; TSO_IN, PF_Ch2RVL
MOV(021) D10019 D13509  ; PF_Ch2RVR
MOV(021) D10020 D13510  ; PF_Ch3RVL
MOV(021) D10021 D13511  ; PF_Ch3RVR
MOV(021) D10022 D13512  ; PF_Ch1NCL
MOV(021) D10023 D13513  ; PF_Ch1NCR
MOV(021) D10024 D13514  ; PF_Ch1NOL
MOV(021) D10025 D13515  ; PF_Ch1NOR
MOV(021) D10026 D13516  ; PF_Ch1CGL
MOV(021) D10027 D13517  ; PF_Ch1CGR
MOV(021) D10028 D13518  ; NC_IN, PF_Ch2NCL
MOV(021) D10029 D13519  ; PF_Ch2NCR
MOV(021) D10030 D13520  ; NO_IN, PF_Ch2NOL
MOV(021) D10031 D13521  ; PF_Ch2NOR
MOV(021) D10032 D13522  ; CG_IN, PF_Ch2CGL
MOV(021) D10033 D13523  ; PF_Ch2CGR
MOV(021) D10034 D13524  ; PF_Ch3NCL
MOV(021) D10035 D13525  ; PF_Ch3NCR
MOV(021) D10036 D13526  ; PF_Ch3NOL
MOV(021) D10037 D13527  ; PF_Ch3NOR
MOV(021) D10038 D13528  ; PF_Ch3CGL
MOV(021) D10039 D13529  ; PF_Ch3CGR
MOV(021) D10040 D13530  ; PF_Ch3TOL
MOV(021) D10041 D13801  ; PF_Ch3TOR

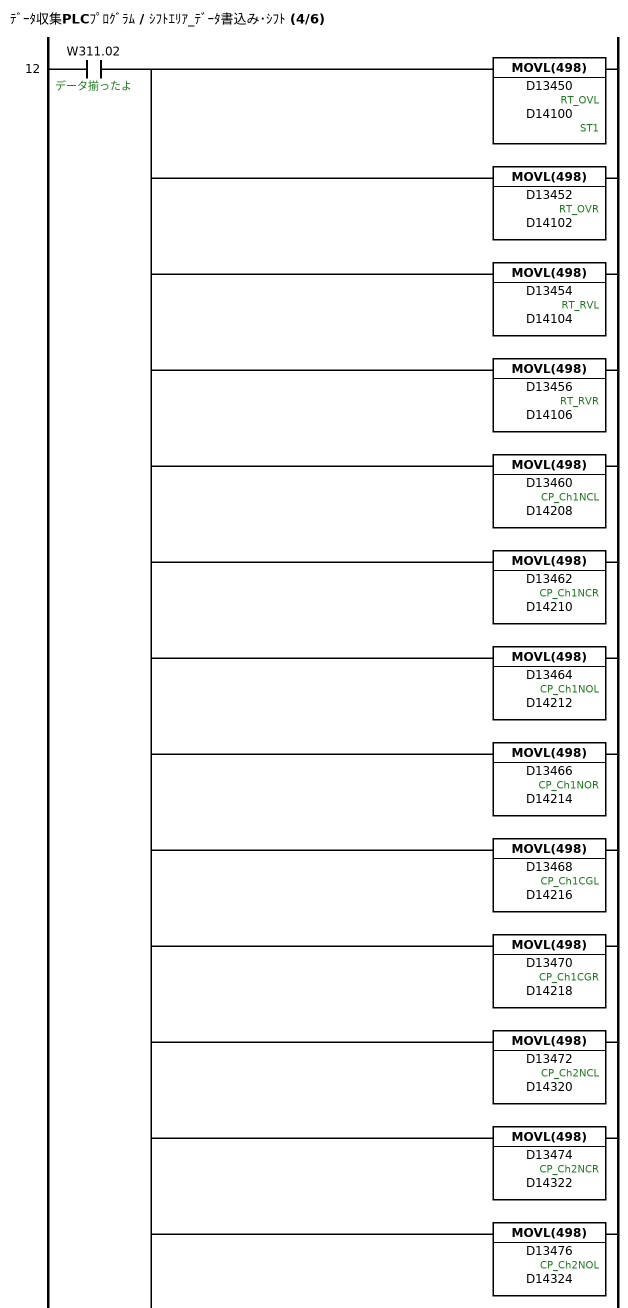

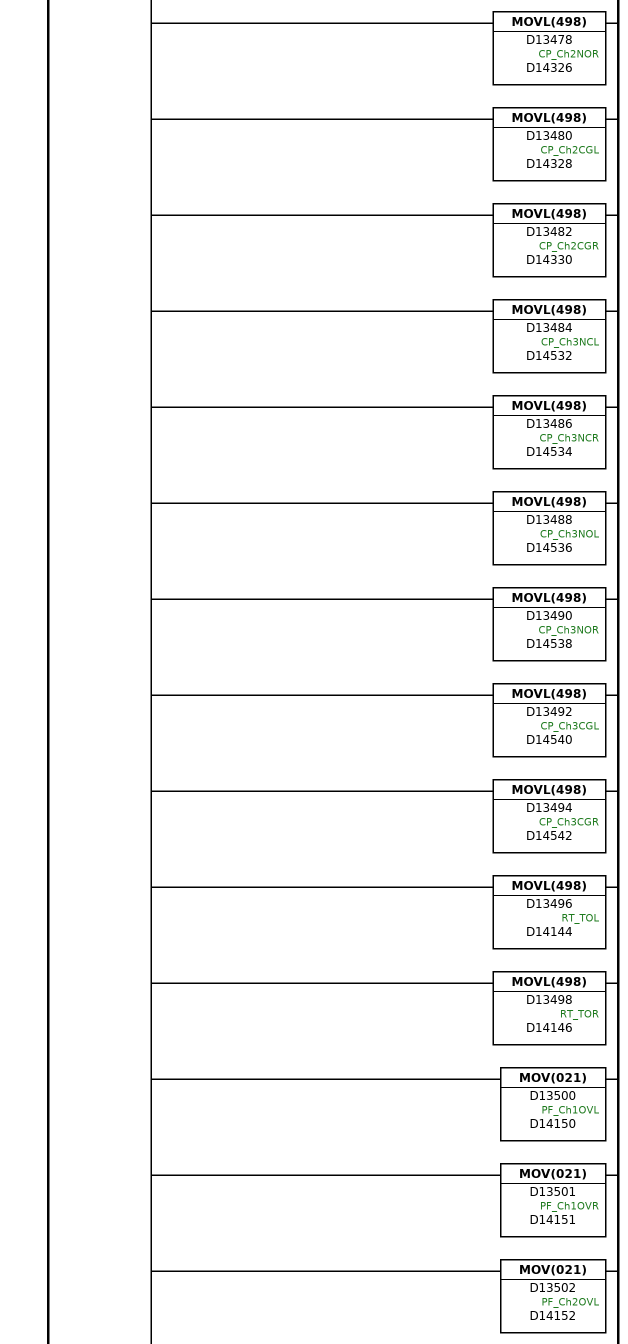

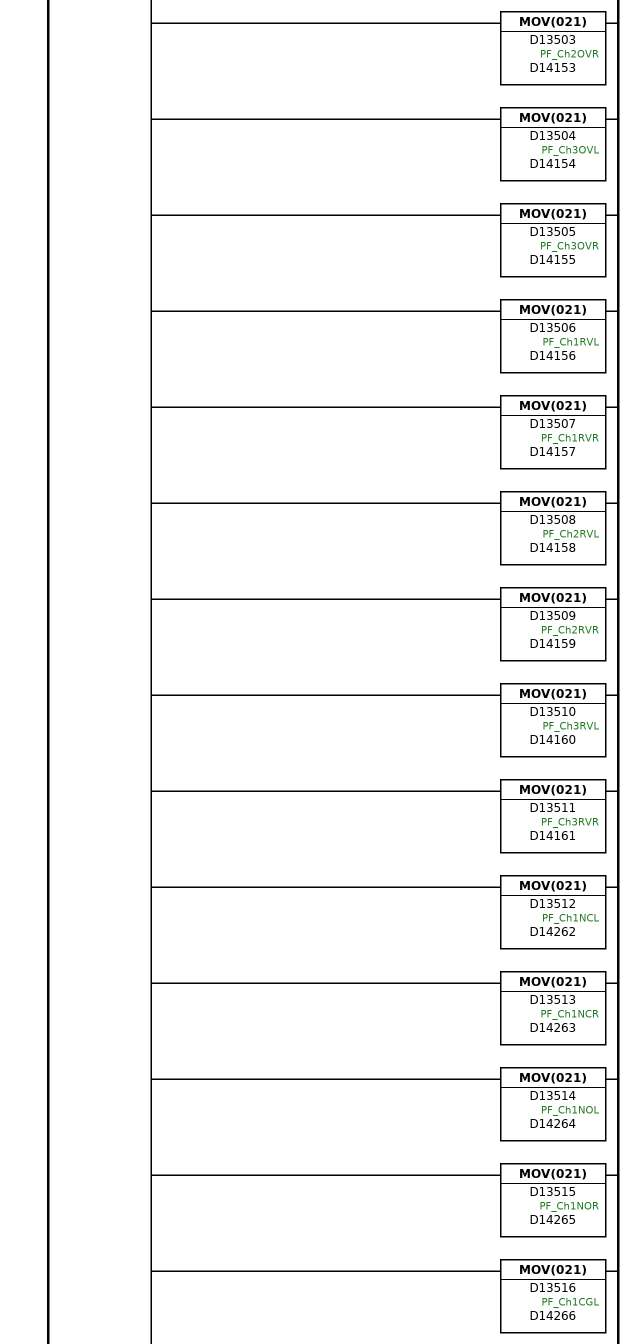

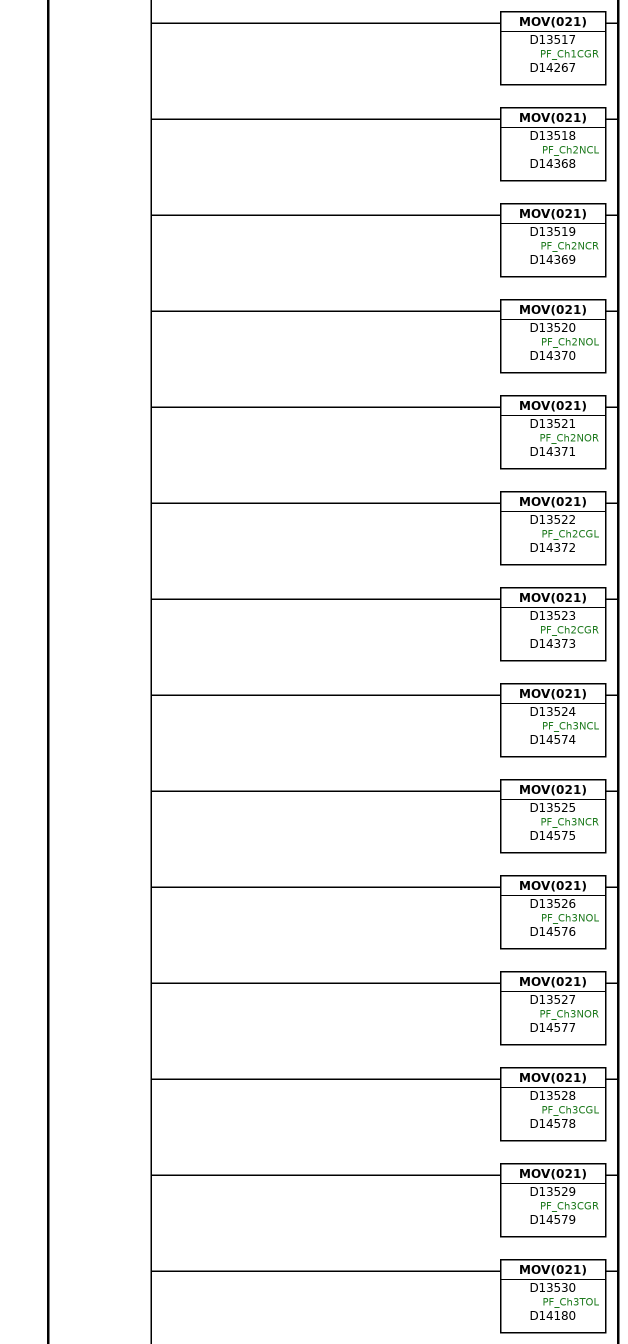

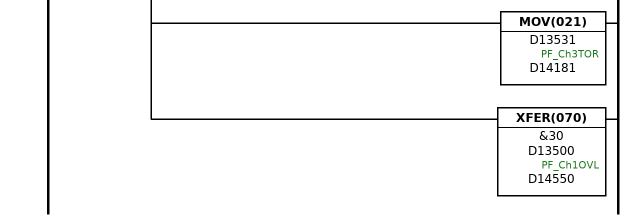
; rung 12
LD W311.02  ; データ揃ったよ
MOVL(498) D13450 D14100  ; RT_OVL, ST1
MOVL(498) D13452 D14102  ; RT_OVR
MOVL(498) D13454 D14104  ; RT_RVL
MOVL(498) D13456 D14106  ; RT_RVR
MOVL(498) D13460 D14208  ; CP_Ch1NCL
MOVL(498) D13462 D14210  ; CP_Ch1NCR
MOVL(498) D13464 D14212  ; CP_Ch1NOL
MOVL(498) D13466 D14214  ; CP_Ch1NOR
MOVL(498) D13468 D14216  ; CP_Ch1CGL
MOVL(498) D13470 D14218  ; CP_Ch1CGR
MOVL(498) D13472 D14320  ; CP_Ch2NCL
MOVL(498) D13474 D14322  ; CP_Ch2NCR
MOVL(498) D13476 D14324  ; CP_Ch2NOL
MOVL(498) D13478 D14326  ; CP_Ch2NOR
MOVL(498) D13480 D14328  ; CP_Ch2CGL
MOVL(498) D13482 D14330  ; CP_Ch2CGR
MOVL(498) D13484 D14532  ; CP_Ch3NCL
MOVL(498) D13486 D14534  ; CP_Ch3NCR
MOVL(498) D13488 D14536  ; CP_Ch3NOL
MOVL(498) D13490 D14538  ; CP_Ch3NOR
MOVL(498) D13492 D14540  ; CP_Ch3CGL
MOVL(498) D13494 D14542  ; CP_Ch3CGR
MOVL(498) D13496 D14144  ; RT_TOL
MOVL(498) D13498 D14146  ; RT_TOR
MOV(021) D13500 D14150  ; PF_Ch1OVL
MOV(021) D13501 D14151  ; PF_Ch1OVR
MOV(021) D13502 D14152  ; PF_Ch2OVL
MOV(021) D13503 D14153  ; PF_Ch2OVR
MOV(021) D13504 D14154  ; PF_Ch3OVL
MOV(021) D13505 D14155  ; PF_Ch3OVR
MOV(021) D13506 D14156  ; PF_Ch1RVL
MOV(021) D13507 D14157  ; PF_Ch1RVR
MOV(021) D13508 D14158  ; PF_Ch2RVL
MOV(021) D13509 D14159  ; PF_Ch2RVR
MOV(021) D13510 D14160  ; PF_Ch3RVL
MOV(021) D13511 D14161  ; PF_Ch3RVR
MOV(021) D13512 D14262  ; PF_Ch1NCL
MOV(021) D13513 D14263  ; PF_Ch1NCR
MOV(021) D13514 D14264  ; PF_Ch1NOL
MOV(021) D13515 D14265  ; PF_Ch1NOR
MOV(021) D13516 D14266  ; PF_Ch1CGL
MOV(021) D13517 D14267  ; PF_Ch1CGR
MOV(021) D13518 D14368  ; PF_Ch2NCL
MOV(021) D13519 D14369  ; PF_Ch2NCR
MOV(021) D13520 D14370  ; PF_Ch2NOL
MOV(021) D13521 D14371  ; PF_Ch2NOR
MOV(021) D13522 D14372  ; PF_Ch2CGL
MOV(021) D13523 D14373  ; PF_Ch2CGR
MOV(021) D13524 D14574  ; PF_Ch3NCL
MOV(021) D13525 D14575  ; PF_Ch3NCR
MOV(021) D13526 D14576  ; PF_Ch3NOL
MOV(021) D13527 D14577  ; PF_Ch3NOR
MOV(021) D13528 D14578  ; PF_Ch3CGL
MOV(021) D13529 D14579  ; PF_Ch3CGR
MOV(021) D13530 D14180  ; PF_Ch3TOL
MOV(021) D13531 D14181  ; PF_Ch3TOR
XFER(070) &30 D13500 D14550  ; PF_Ch1OVL

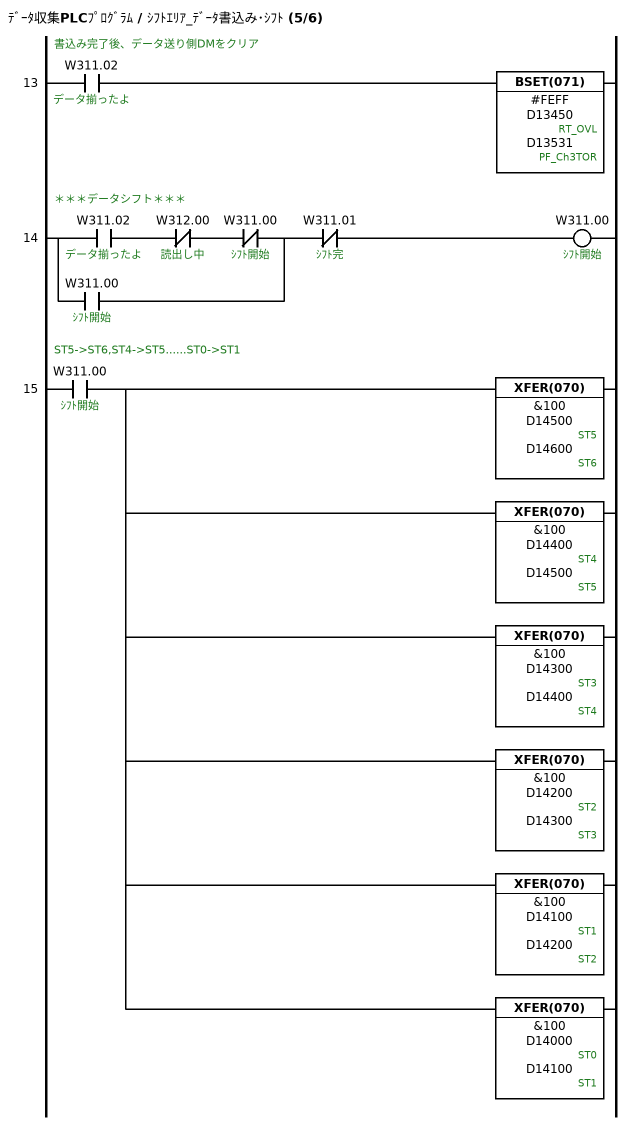
; rung 13: 書込み完了後、データ送り側DMをクリア
LD W311.02  ; データ揃ったよ
BSET(071) #FEFF D13450 D13531  ; RT_OVL, PF_Ch3TOR
; rung 14: ＊＊＊データシフト＊＊＊
LD W311.02  ; データ揃ったよ
ANDNOT W312.00  ; 読出し中
ANDNOT W311.00  ; ｼﾌﾄ開始
OR W311.00  ; ｼﾌﾄ開始
ANDNOT W311.01  ; ｼﾌﾄ完
OUT W311.00  ; ｼﾌﾄ開始
; rung 15: ST5->ST6,ST4->ST5......ST0->ST1
LD W311.00  ; ｼﾌﾄ開始
XFER(070) &100 D14500 D14600  ; ST5, ST6
XFER(070) &100 D14400 D14500  ; ST4, ST5
XFER(070) &100 D14300 D14400  ; ST3, ST4
XFER(070) &100 D14200 D14300  ; ST2, ST3
XFER(070) &100 D14100 D14200  ; ST1, ST2
XFER(070) &100 D14000 D14100  ; ST0, ST1

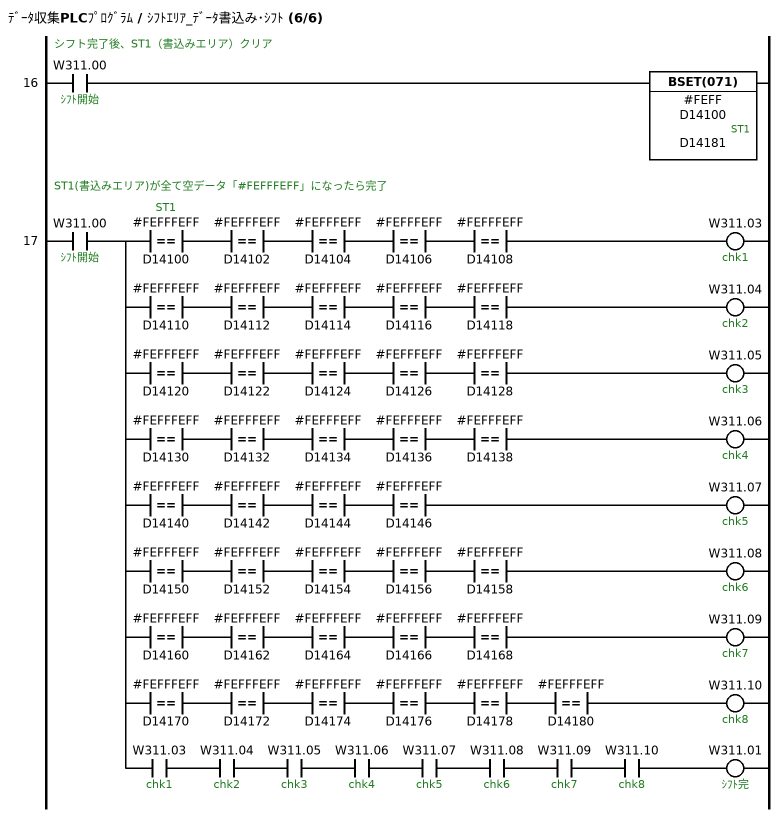
; rung 16: シフト完了後、ST1（書込みエリア）クリア
LD W311.00  ; ｼﾌﾄ開始
BSET(071) #FEFF D14100 D14181  ; ST1
; rung 17: ST1(書込みエリア)が全て空データ「#FEFFFEFF」になったら完了
LD W311.00  ; ｼﾌﾄ開始
OUT TR0
AND=L(301) #FEFFFEFF D14100  ; ST1
AND=L(301) #FEFFFEFF D14102
AND=L(301) #FEFFFEFF D14104
AND=L(301) #FEFFFEFF D14106
AND=L(301) #FEFFFEFF D14108
OUT W311.03  ; chk1
LD TR0
AND=L(301) #FEFFFEFF D14110
AND=L(301) #FEFFFEFF D14112
AND=L(301) #FEFFFEFF D14114
AND=L(301) #FEFFFEFF D14116
AND=L(301) #FEFFFEFF D14118
OUT W311.04  ; chk2
LD TR0
AND=L(301) #FEFFFEFF D14120
AND=L(301) #FEFFFEFF D14122
AND=L(301) #FEFFFEFF D14124
AND=L(301) #FEFFFEFF D14126
AND=L(301) #FEFFFEFF D14128
OUT W311.05  ; chk3
LD TR0
AND=L(301) #FEFFFEFF D14130
AND=L(301) #FEFFFEFF D14132
AND=L(301) #FEFFFEFF D14134
AND=L(301) #FEFFFEFF D14136
AND=L(301) #FEFFFEFF D14138
OUT W311.06  ; chk4
LD TR0
AND=L(301) #FEFFFEFF D14140
AND=L(301) #FEFFFEFF D14142
AND=L(301) #FEFFFEFF D14144
AND=L(301) #FEFFFEFF D14146
OUT W311.07  ; chk5
LD TR0
AND=L(301) #FEFFFEFF D14150
AND=L(301) #FEFFFEFF D14152
AND=L(301) #FEFFFEFF D14154
AND=L(301) #FEFFFEFF D14156
AND=L(301) #FEFFFEFF D14158
OUT W311.08  ; chk6
LD TR0
AND=L(301) #FEFFFEFF D14160
AND=L(301) #FEFFFEFF D14162
AND=L(301) #FEFFFEFF D14164
AND=L(301) #FEFFFEFF D14166
AND=L(301) #FEFFFEFF D14168
OUT W311.09  ; chk7
LD TR0
AND=L(301) #FEFFFEFF D14170
AND=L(301) #FEFFFEFF D14172
AND=L(301) #FEFFFEFF D14174
AND=L(301) #FEFFFEFF D14176
AND=L(301) #FEFFFEFF D14178
AND=L(301) #FEFFFEFF D14180
OUT W311.10  ; chk8
LD TR0
AND W311.03  ; chk1
AND W311.04  ; chk2
AND W311.05  ; chk3
AND W311.06  ; chk4
AND W311.07  ; chk5
AND W311.08  ; chk6
AND W311.09  ; chk7
AND W311.10  ; chk8
OUT W311.01  ; ｼﾌﾄ完

### Section ｼﾌﾄｴﾘｱ_ﾃﾞｰﾀ読出し

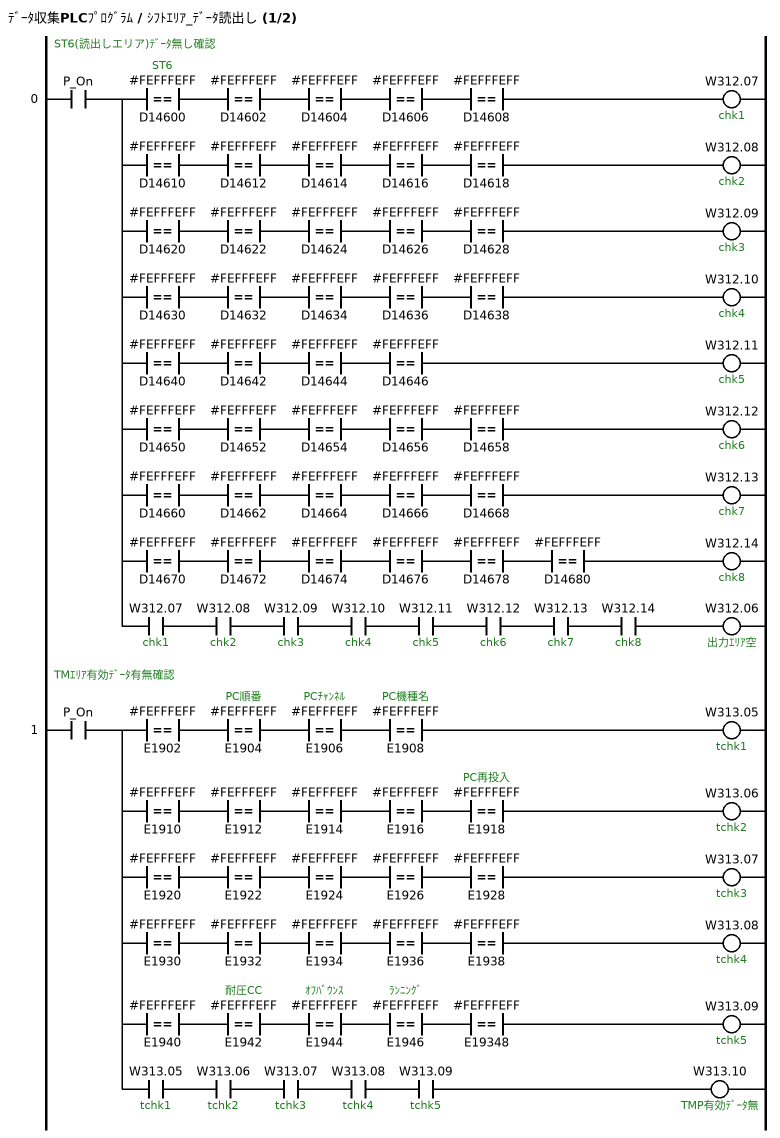
; rung 0: ST6(読出しエリア)ﾃﾞｰﾀ無し確認
LD P_On
OUT TR0
AND=L(301) #FEFFFEFF D14600  ; ST6
AND=L(301) #FEFFFEFF D14602
AND=L(301) #FEFFFEFF D14604
AND=L(301) #FEFFFEFF D14606
AND=L(301) #FEFFFEFF D14608
OUT W312.07  ; chk1
LD TR0
AND=L(301) #FEFFFEFF D14610
AND=L(301) #FEFFFEFF D14612
AND=L(301) #FEFFFEFF D14614
AND=L(301) #FEFFFEFF D14616
AND=L(301) #FEFFFEFF D14618
OUT W312.08  ; chk2
LD TR0
AND=L(301) #FEFFFEFF D14620
AND=L(301) #FEFFFEFF D14622
AND=L(301) #FEFFFEFF D14624
AND=L(301) #FEFFFEFF D14626
AND=L(301) #FEFFFEFF D14628
OUT W312.09  ; chk3
LD TR0
AND=L(301) #FEFFFEFF D14630
AND=L(301) #FEFFFEFF D14632
AND=L(301) #FEFFFEFF D14634
AND=L(301) #FEFFFEFF D14636
AND=L(301) #FEFFFEFF D14638
OUT W312.10  ; chk4
LD TR0
AND=L(301) #FEFFFEFF D14640
AND=L(301) #FEFFFEFF D14642
AND=L(301) #FEFFFEFF D14644
AND=L(301) #FEFFFEFF D14646
OUT W312.11  ; chk5
LD TR0
AND=L(301) #FEFFFEFF D14650
AND=L(301) #FEFFFEFF D14652
AND=L(301) #FEFFFEFF D14654
AND=L(301) #FEFFFEFF D14656
AND=L(301) #FEFFFEFF D14658
OUT W312.12  ; chk6
LD TR0
AND=L(301) #FEFFFEFF D14660
AND=L(301) #FEFFFEFF D14662
AND=L(301) #FEFFFEFF D14664
AND=L(301) #FEFFFEFF D14666
AND=L(301) #FEFFFEFF D14668
OUT W312.13  ; chk7
LD TR0
AND=L(301) #FEFFFEFF D14670
AND=L(301) #FEFFFEFF D14672
AND=L(301) #FEFFFEFF D14674
AND=L(301) #FEFFFEFF D14676
AND=L(301) #FEFFFEFF D14678
AND=L(301) #FEFFFEFF D14680
OUT W312.14  ; chk8
LD TR0
AND W312.07  ; chk1
AND W312.08  ; chk2
AND W312.09  ; chk3
AND W312.10  ; chk4
AND W312.11  ; chk5
AND W312.12  ; chk6
AND W312.13  ; chk7
AND W312.14  ; chk8
OUT W312.06  ; 出力ｴﾘｱ空
; rung 1: TMｴﾘｱ有効ﾃﾞｰﾀ有無確認
LD P_On
OUT TR0
AND=L(301) #FEFFFEFF E1902
AND=L(301) #FEFFFEFF E1904  ; PC順番
AND=L(301) #FEFFFEFF E1906  ; PCﾁｬﾝﾈﾙ
AND=L(301) #FEFFFEFF E1908  ; PC機種名
OUT W313.05  ; tchk1
LD TR0
AND=L(301) #FEFFFEFF E1910
AND=L(301) #FEFFFEFF E1912
AND=L(301) #FEFFFEFF E1914
AND=L(301) #FEFFFEFF E1916
AND=L(301) #FEFFFEFF E1918  ; PC再投入
OUT W313.06  ; tchk2
LD TR0
AND=L(301) #FEFFFEFF E1920
AND=L(301) #FEFFFEFF E1922
AND=L(301) #FEFFFEFF E1924
AND=L(301) #FEFFFEFF E1926
AND=L(301) #FEFFFEFF E1928
OUT W313.07  ; tchk3
LD TR0
AND=L(301) #FEFFFEFF E1930
AND=L(301) #FEFFFEFF E1932
AND=L(301) #FEFFFEFF E1934
AND=L(301) #FEFFFEFF E1936
AND=L(301) #FEFFFEFF E1938
OUT W313.08  ; tchk4
LD TR0
AND=L(301) #FEFFFEFF E1940
AND=L(301) #FEFFFEFF E1942  ; 耐圧CC
AND=L(301) #FEFFFEFF E1944  ; ｵﾌﾊﾞｳﾝｽ
AND=L(301) #FEFFFEFF E1946  ; ﾗﾝﾆﾝｸﾞ
AND=L(301) #FEFFFEFF E19348
OUT W313.09  ; tchk5
LD TR0
AND W313.05  ; tchk1
AND W313.06  ; tchk2
AND W313.07  ; tchk3
AND W313.08  ; tchk4
AND W313.09  ; tchk5
OUT W313.10  ; TMP有効ﾃﾞｰﾀ無

